text list "AlarmList": 1000 'F01000 - Внутрішня програмна помилка'; 1001 'F01001 - Виняток операції з плаваючою комою'; 1002 'F01002 - Внутрішня програмна помилка'; 1003 'F01003 - Затримка квитування під час доступу до пам’яті'; 1004 'N01004 (F, A) - Внутрішня програмна помилка'; 1005 'F01005 - Не вдалося завантажити прошивку компонента DRIVE-CLiQ'; 1006 'A01006 - Потрібне оновлення прошивки компонента DRIVE-CLiQ'; 1007 'A01007 - Потрібне повторне увімкнення живлення компонента DRIVE-CLiQ'; 1009 'A01009 (N) - CU: Перегрів модуля керування'; 1010 'F01010 - Невідомий тип приводу'; 1011 'F01011 (N) - Завантаження перервано'; 1012 'F01012 (N) - Помилка перетворення проєкту'; 1013 'A01013 - CU: Досягнуто або перевищено граничний ресурс вентилятора'; 1014 'F01014 - Топологія: змінено властивість компонента DRIVE-CLiQ'; 1015 'F01015 - Внутрішня програмна помилка'; 1016 'A01016 (F) - Змінено версію прошивки'; 1017 'A01017 - Змінено списки компонентів'; 1020 'A01020 - Не вдалося записати дані на RAM-диск'; 1023 'F01023 - Внутрішній програмний тайм-аут'; 1030 'F01030 - Відсутній сигнал справності головного керування'; 1031 'F01031 - Відсутній сигнал справності команди OFF у режимі REMOTE'; 1032 'A01032 (F) - ACX: Необхідно зберегти всі параметри'; 1033 'F01033 - Перемикання одиниць: некоректне опорне значення параметра'; 1034 'F01034 - Перемикання одиниць: не вдалося обчислити значення параметрів після зміни опорного значення'; 1035 'A01035 (F) - ACX: Пошкоджено файл резервної копії параметрів'; 1036 'F01036 (A) - ACX: Відсутній файл резервної копії параметрів'; 1038 'F01038 (A) - ACX: Не вдалося завантажити файл резервної копії параметрів'; 1039 'F01039 (A) - ACX: Не вдалося записати файл резервної копії параметрів'; 1040 'F01040 - Збережіть налаштування параметрів і виконайте повторне увімкнення живлення'; 1041 'F01041 - Потрібно зберегти параметри'; 1042 'F01042 - Помилка параметрів під час завантаження проєкту'; 1043 'F01043 - Критична помилка під час завантаження проєкту'; 1044 'F01044 - CU: Помилка описових даних'; 1045 'A01045 - CU: Некоректні конфігураційні дані'; 1049 'A01049 - CU: Не вдалося записати дані у файл'; 1050 'F01050 - Карта пам’яті несумісна з пристроєм'; 1054 'F01054 - CU: Перевищено системне обмеження'; 1055 'F01055 - CU: Внутрішня помилка (SYNO порту та прикладної програми не збігаються)'; 1056 'F01056 - CU: Внутрішня помилка (тактовий цикл групи параметрів уже призначено інакше)'; 1057 'F01057 - CU: Внутрішня помилка (інший тип DRIVE-CLiQ для підлеглого пристрою)'; 1058 'F01058 - CU: Внутрішня помилка (у топології відсутній підлеглий пристрій)'; 1059 'F01059 - CU: Внутрішня помилка (порт не існує)'; 1060 'F01060 - CU: Внутрішня помилка (група параметрів недоступна)'; 1061 'F01061 - CU: Внутрішня помилка (невідома прикладна програма)'; 1063 'F01063 - CU: Внутрішня помилка (PDM)'; 1064 'A01064 (F) - CU: Внутрішня помилка (CRC)'; 1068 'F01068 - CU: Переповнення пам’яті даних'; 1069 'A01069 - Несумісність резервної копії параметрів і пристрою'; 1070 'F01070 - Виконується завантаження проєкту/прошивки на карту пам’яті'; 1072 'F01072 - Карту пам’яті відновлено з резервної копії'; 1073 'A01073 (N) - Для резервної копії на карті пам’яті потрібне повторне увімкнення живлення'; 1082 'F01082 - Помилка параметрів під час увімкнення з резервної копії даних'; 1097 'A01097 (N) - Сервер NTP недоступний'; 1099 'A01099 (N) - Перевищено допуск синхронізації UTC'; 1100 'A01100 - CU: Карту пам’яті вилучено'; 1105 'F01105 (A) - CU: Недостатньо пам’яті'; 1106 'F01106 - CU: Недостатньо пам’яті'; 1107 'F01107 - CU: Не вдалося зберегти дані на карту пам’яті'; 1110 'F01110 - CU: До одного модуля керування підключено більше одного SINAMICS G'; 1111 'F01111 - CU: Змішана робота приводних модулів не допускається'; 1112 'F01112 - CU: Використання силового модуля не допускається'; 1120 'F01120 (A) - Не вдалося ініціалізувати термінал'; 1122 'F01122 (A) - Частота на вході вимірювального щупа занадто висока'; 1123 'F01123 - Силовий модуль не підтримує дискретні входи/виходи'; 1150 'F01150 - CU: Перевищено кількість екземплярів типу об’єкта приводу'; 1151 'F01151 - CU: Перевищено кількість об’єктів приводу заданої категорії'; 1152 'F01152 - CU: Некоректна комбінація типів об’єктів приводу'; 1200 'F01200 - CU: Внутрішня програмна помилка керування часовими квантами'; 1205 'F01205 - CU: Переповнення часового кванта'; 1221 'F01221 - CU: Базовий тактовий цикл занадто малий'; 1222 'F01222 - CU: Базовий тактовий цикл занадто малий (недостатньо часу на обробку зв’язку)'; 1223 'A01223 - CU: Некоректний час дискретизації'; 1224 'A01224 - CU: Некоректна частота імпульсів'; 1250 'F01250 - CU: Некоректні дані CU-EEPROM, доступні лише для читання'; 1251 'A01251 - CU: Некоректні дані читання/запису CU-EEPROM'; 1255 'F01255 - CU: Помилка даних EEPROM плати розширення, доступних лише для читання'; 1256 'A01256 - CU: Помилка даних читання/запису EEPROM плати розширення'; 1260 'F01260 - Програмне забезпечення не активоване'; 1275 'F01275 - Помилка опису обладнання'; 1276 'A01276 - Опис обладнання не повністю сумісний'; 1302 'A01302 - Помилка у трасуванні компонента'; 1303 'F01303 - Компонент виконує не підтримка потрібно функція'; 1304 'A01304 (F) - Версія прошивки компонента DRIVE-CLiQ застаріла'; 1305 'F01305 - Топологія: відсутній номер компонента'; 1306 'A01306 - Виконується оновлення прошивки компонента DRIVE-CLiQ'; 1314 'A01314 - Топологія: Компонент повинен не бути наявний'; 1317 'A01317 (N) - Деактивовано компонент повторно наявний'; 1318 'A01318 - BICO: наявні деактивовані міжз’єднання'; 1319 'A01319 - Встановлений компонент не ініціалізовано'; 1320 'A01320 - Топологія: номер об’єкта приводу відсутній у конфігурації'; 1321 'A01321 - Топологія: номер об’єкта приводу відсутній у конфігурації'; 1322 'A01322 - Топологія: номер об’єкта приводу двічі присутній у конфігурації'; 1323 'A01323 - Топологія: створено більше двох часткових списків'; 1324 'A01324 - Топологія: номер фіктивного об’єкта приводу створено некоректно'; 1325 'F01325 - Топологія: номер компонента відсутній у цільовій топології'; 1330 'A01330 - Топологія: швидке введення в експлуатацію неможливе'; 1331 'A01331 - Топологія: щонайменше один компонент не призначено об’єкту приводу'; 1340 'F01340 - Топологія: на одній лінії забагато компонентів'; 1341 'F01341 - Топологія: перевищено максимальну кількість компонентів DRIVE-CLiQ'; 1354 'F01354 - Топологія: фактична топологія містить неприпустимий компонент'; 1355 'F01355 - Топологія: Фактичний топологія змінено'; 1356 'F01356 - Топологія: виявлено несправний компонент DRIVE-CLiQ'; 1357 'F01357 - Топологія: на лінії DRIVE-CLiQ ідентифіковано два модулі керування'; 1358 'A01358 - Топологія: термінування лінії недоступне'; 1359 'F01359 - Топологія: продуктивність DRIVE-CLiQ недостатня'; 1360 'F01360 - Топологія: Фактичний топологія не допустимий'; 1361 'A01361 - Топологія: фактична топологія містить компоненти SINUMERIK і SIMOTION'; 1362 'A01362 - Топологія: порушено правило(а) топології'; 1375 'F01375 - Топологія: між двома компонентами дубльовано з’єднання'; 1380 'F01380 - Топологія: Фактичний топологія EEPROM несправний'; 1381 'A01381 - Топологія: силовий модуль встановлено некоректно'; 1382 'A01382 - Топологія: модуль датчика встановлено некоректно'; 1383 'A01383 - Топологія: термінальний модуль встановлено некоректно'; 1384 'A01384 - Топологія: модуль-концентратор DRIVE-CLiQ встановлено некоректно'; 1385 'A01385 - Топологія: модуль розширення контролера встановлено некоректно'; 1386 'A01386 - Топологія: компонент DRIVE-CLiQ встановлено некоректно'; 1389 'A01389 - Топологія: двигун із DRIVE-CLiQ встановлено некоректно'; 1416 'A01416 - Топологія: додатково встановлено компонент'; 1420 'A01420 - Топологія: Компонент інший'; 1425 'A01425 - Топологія: інший серійний номер'; 1428 'A01428 - Топологія: використано некоректне з’єднання'; 1451 'F01451 - Топологія: цільова топологія некоректна'; 1481 'A01481 (N) - Топологія: силовий модуль не підключено'; 1482 'A01482 - Топологія: модуль датчика не підключено'; 1483 'A01483 - Топологія: термінальний модуль не підключено'; 1484 'A01484 - Топологія: модуль-концентратор DRIVE-CLiQ не підключено'; 1485 'A01485 - Топологія: модуль розширення контролера не підключено'; 1486 'A01486 - Топологія: компонент DRIVE-CLiQ не підключено'; 1487 'A01487 - Топологія: компонент у слоті опцій не встановлено'; 1489 'A01489 - Топологія: двигун із DRIVE-CLiQ не підключено'; 1507 'A01507 (F, N) - BICO: наявні міжз’єднання з неактивними об’єктами'; 1508 'A01508 - BICO: перевищено кількість міжз’єднань з неактивними об’єктами'; 1510 'F01510 - BICO: джерело сигналу не має типу FLOAT'; 1511 'F01511 (A) - BICO: міжз’єднання з різними масштабуваннями'; 1512 'F01512 - BICO: масштабування недоступне'; 1513 'F01513 (N, A) - BICO: міжз’єднання між об’єктами приводу з різними масштабуваннями'; 1514 'A01514 (F) - BICO: помилка запису під час повторного з’єднання'; 1515 'F01515 (A) - BICO: запис до параметра не допускається, оскільки активне головне керування'; 1590 'A01590 (F) - Привід: перевищено інтервал технічного обслуговування двигуна'; 1600 'F01600 - SI P1 (CU): Ініційовано зупинку A'; 1611 'F01611 (A) - SI P1 (CU): Несправність у каналі контролю'; 1612 'F01612 - SI P1 (CU): Різні STO-входи силових модулів, підключених паралельно'; 1620 'N01620 (F, A) - SI P1 (CU): Безпечне вимкнення крутного моменту активний'; 1621 'N01621 (F, A) - SI P1 (CU): Активна безпечна зупинка 1'; 1625 'F01625 - SI P1 (CU): Помилка сигналу справності в даних безпеки'; 1630 'F01630 - SI P1 (CU): Гальмо керування помилка'; 1631 'A01631 (F, N) - SI P1 (CU): Конфігурація гальма утримання двигуна/SBC непрактична'; 1632 'F01632 - SI P1 (CU): Помилка сигналу керування/зворотного зв’язку запірного клапана'; 1640 'F01640 (N, A) - SI P1 (CU): Виявлено заміну компонента; потрібні квитування та збереження'; 1641 'F01641 (N, A) - SI P1 (CU): Виявлено заміну компонента; потрібне збереження'; 1649 'F01649 - SI P1 (CU): Внутрішня програмна помилка'; 1650 'F01650 - SI P1 (CU): Потрібне приймальне випробування'; 1651 'F01651 - SI P1 (CU): Не вдалося синхронізувати часові кванти безпеки'; 1652 'F01652 - SI P1 (CU): неприпустимий тактовий цикл контролю'; 1653 'F01653 - SI P1 (CU): PROFIBUS/PROFINET конфігурація помилка'; 1654 'A01654 (F, N) - SI P1 (CU): Відхилення конфігурації PROFIsafe'; 1655 'F01655 - SI P1 (CU): Узгодьте функції контролю'; 1656 'F01656 - SI CU: Помилка каналу 2 контролю параметрів'; 1657 'F01657 - SI P1 (CU): Некоректний номер телеграми PROFIsafe'; 1658 'F01658 - SI P1 (CU): Номери телеграм PROFIsafe відрізняються'; 1659 'F01659 - SI P1 (CU): Запит на запис параметра відхилено'; 1660 'F01660 - SI P1 (CU): Функції, пов’язані з безпекою, не підтримуються'; 1661 'F01661 - SI P1 (CU): Активна симуляція входів безпеки'; 1663 'F01663 - SI P1 (CU): Копіювання параметрів SI відхилено'; 1664 'F01664 - SI P1 (CU): Відсутнє автоматичне оновлення прошивки'; 1665 'F01665 - SI P1 (CU): Система несправна'; 1666 'A01666 (F) - SI Motion P1 (CU): Постійний сигнал «1» на F-DI для безпечного квитування'; 1669 'A01669 (F, N) - SI Motion: Несприятлива комбінація двигуна та силового модуля'; 1670 'F01670 - SI Motion: Некоректна параметризація модуля датчика'; 1671 'F01671 - SI Motion: Помилка параметризації енкодера'; 1672 'F01672 - SI P1 (CU): Програмне/апаратне забезпечення моторного модуля несумісне'; 1673 'F01673 - SI Motion: Програмне/апаратне забезпечення модуля датчика несумісне'; 1674 'F01674 - SI Motion P1 (CU): Функція безпеки не підтримується телеграмою PROFIsafe'; 1675 'F01675 - SI Motion P1: Налаштування у контролері PROFIBUS/PROFINET не допускаються'; 1679 'F01679 - SI CU: Змінено налаштування параметрів безпеки та топологію; потрібен теплий перезапуск/POWER ON'; 1680 'F01680 - SI Motion P1 (CU): Помилка контрольної суми функцій контролю безпеки'; 1681 'F01681 - SI Motion P1 (CU): Некоректне значення параметра'; 1682 'F01682 - SI Motion P1 (CU): Функція контролю не підтримується'; 1683 'F01683 - SI Motion P1 (CU): Відсутній дозвіл SOS/SLS'; 1684 'F01684 - SI Motion P1 (CU): Граничні значення безпечно обмеженого положення переплутано'; 1685 'F01685 - SI Motion P1 (CU): Граничне значення безпечно обмеженої швидкості занадто високе'; 1686 'F01686 - SI Motion: Некоректна параметризація кулачкового положення'; 1687 'F01687 - SI Motion: Некоректна параметризація модульного значення SCA (SN)'; 1688 'F01688 - SI Motion CU: Фактичний значення синхронізація не допустимий'; 1689 'C01689 - SI Motion: Вісь повторно сконфігуровано'; 1690 'F01690 - SI Motion: Помилка збереження даних у NVRAM'; 1691 'A01691 (F) - SI Motion: Значення Ti та To непридатні для циклу DP'; 1692 'F01692 - SI Motion P1 (CU): Значення параметра не допускається для режиму без енкодера'; 1693 'A01693 (F) - SI P1 (CU): Змінено налаштування параметрів безпеки; потрібен теплий перезапуск/повторне увімкнення живлення'; 1694 'F01694 (A) - SI Motion CU: Версія прошивки моторного/гідравлічного модуля старіша за версію модуля керування'; 1695 'A01695 (F) - SI Motion: Модуль датчика замінено'; 1696 'A01696 (F) - SI Motion: Під час завантаження вибрано тестову зупинку для функцій контролю руху'; 1697 'A01697 (F) - SI Motion: Потрібна тестова зупинка для функцій контролю руху'; 1698 'A01698 (F) - SI P1 (CU): Активний режим введення в експлуатацію'; 1699 'A01699 (F) - SI P1 (CU): Потрібна тестова зупинка для STO'; 1700 'C01700 - SI Motion P1 (CU): Ініційовано зупинку A'; 1701 'C01701 - SI Motion P1 (CU): Ініційовано зупинку B'; 1706 'C01706 - SI Motion P1 (CU): Перевищено обмеження SAM/SBR'; 1707 'C01707 - SI Motion P1 (CU): Перевищено допуск для безпечної робочої зупинки'; 1708 'C01708 - SI Motion P1 (CU): Ініційовано зупинку C'; 1709 'C01709 - SI Motion P1 (CU): Ініційовано зупинку D'; 1710 'C01710 - SI Motion P1 (CU): Ініційовано зупинку E'; 1711 'C01711 - SI Motion P1 (CU): Несправність у каналі контролю'; 1712 'C01712 - SI Motion P1 (CU): Несправність обробки F-IO'; 1714 'C01714 - SI Motion P1 (CU): Безпечно обмежена швидкість перевищено'; 1715 'C01715 - SI Motion P1 (CU): Безпечно обмежене положення перевищено'; 1716 'C01716 - SI Motion P1 (CU): Перевищено допуск для безпечного напрямку руху'; 1717 'C01717 - SI Motion P1 (CU): Перевищено обмеження SLA'; 1730 'C01730 - SI Motion P1 (CU): Некоректний опорний блок для динамічної безпечно обмеженої швидкості'; 1745 'C01745 - SI Motion P1 (CU): Перевірка гальмівного моменту для тесту гальма'; 1750 'C01750 - SI Motion P1 (CU): Апаратна несправність енкодера, важливого для безпеки'; 1751 'C01751 - SI Motion P1 (CU): Несправність перевірки ефективності енкодера, важливого для безпеки'; 1752 'C01752 - SI Motion P1 (CU): Некоректне референтне положення'; 1770 'C01770 - SI Motion P1 (CU): Помилка розбіжності відмовобезпечних входів/виходів'; 1772 'A01772 - SI Motion P1 (CU): Виконується тестова зупинка для відмовобезпечних дискретних виходів'; 1773 'F01773 - SI Motion P1 (CU): Помилка тестової зупинки відмовобезпечного дискретного виходу'; 1774 'A01774 - SI Motion P1 (CU): Потрібна тестова зупинка для відмовобезпечних дискретних виходів'; 1780 'A01780 - За вибору SBT гальмо замкнене'; 1781 'A01781 - Перевищено час розгальмовування гальма SBT'; 1782 'A01782 - SBT гальмо тест некоректний керування'; 1783 'A01783 - Перевищено час загальмовування гальма SBT'; 1784 'A01784 - Тест гальма SBT скасовано через несправність'; 1785 'A01785 - Помилка конфігурації тесту гальма SBT'; 1786 'F01786 - Змінено джерело сигналу SCC'; 1787 'F01787 - Інший тип двигуна SBT'; 1788 'A01788 - SI: Автоматична тестова зупинка очікує скасування вибору STO через функції контролю руху'; 1789 'A01789 - SI: Автоматична тестова зупинка та тест гальма не допускаються, коли вибрано тестову зупинку'; 1794 'A01794 (N) - SI Motion: Перевірка модульного значення для безпечного положення через PROFIsafe'; 1795 'A01795 - SI Motion P1 (CU): Перевищено час очікування після виходу зі скасування безпечних імпульсів'; 1796 'A01796 (F, N) - SI P1 (CU): Очікування зв’язку'; 1797 'C01797 - SI Motion P1 (CU): Вісь не пройшла безпечне реферування'; 1798 'C01798 - SI Motion P1 (CU): Тест зупинка для рух контроль функції виконується'; 1799 'C01799 - SI Motion P1 (CU): Приймальне тест режим активний'; 1800 'F01800 (A) - DRIVE-CLiQ: помилка обладнання/конфігурації'; 1839 'A01839 - Діагностика DRIVE-CLiQ: несправність кабелю до компонента'; 1840 'A01840 - SMI: Компонент виявлено без Дані двигуна'; 1900 'A01900 (F) - PB/PN: Конфігурація Помилка телеграми'; 1902 'A01902 - PB/PN: параметризація синхронної роботи за тактовим циклом не допускається'; 1903 'A01903 (F) - COMM INT: Приймання конфігурація дані некоректний'; 1910 'F01910 (N, A) - Польова шина: тайм-аут заданого значення'; 1911 'F01911 (N, A) - PB/PN: відмова тактового циклу синхронної роботи'; 1912 'F01912 (N, A) - PB/PN: відмова сигналу справності синхронної роботи за тактовим циклом'; 1913 'F01913 (N, A) - COMM INT: закінчився контрольний час сигналу справності'; 1914 'F01914 (N, A) - COMM INT: Контроль час конфігурація закінчився'; 1915 'F01915 (N, A) - PB/PN: відмова сигналу справності синхронної роботи за тактовим циклом, об’єкт приводу 1'; 1920 'A01920 (F) - PROFIBUS: перервано циклічне з’єднання'; 1921 'A01921 (F) - PROFIBUS: приймання заданих значень після To'; 1925 'A01925 (F) - Modbus TCP: з’єднання перервано'; 1930 'A01930 - PB/PN: час дискретизації регулятора струму не дорівнює синхронному тактовому циклу'; 1931 'A01931 - PB/PN: час дискретизації регулятора швидкості не дорівнює синхронному тактовому циклу'; 1932 'A01932 - PB/PN: відсутня синхронізація тактового циклу для DSC'; 1940 'A01940 - PB/PN: синхронізм тактового циклу не досягнуто'; 1941 'A01941 - PB/PN: відсутній сигнал тактового циклу під час встановлення зв’язку по шині'; 1943 'A01943 - PB/PN: помилка сигналу тактового циклу під час встановлення зв’язку по шині'; 1944 'A01944 - PB/PN: синхронізм сигналу справності не досягнуто'; 1945 'A01945 - PROFIBUS: З’єднання до Видавець не вдалося виконати'; 1946 'F01946 (A) - PROFIBUS: з’єднання з видавцем перервано'; 1950 'F01950 (N, A) - PB/PN: не вдалося синхронізувати синхронну роботу за тактовим циклом'; 1951 'F01951 - CU SYNC: відсутній тактовий цикл прикладної синхронізації'; 1952 'F01952 - CU DRIVE-CLiQ: синхронізація компонента не підтримується'; 1953 'A01953 - CU SYNC: синхронізацію не завершено'; 1954 'F01954 - CU DRIVE-CLiQ: не вдалося виконати синхронізацію'; 1955 'A01955 - CU DRIVE-CLiQ: синхронізацію об’єкта приводу не завершено'; 1970 'A01970 - CBExx: циклічне з’єднання перервано'; 1971 'A01971 - CBExx: перевищено максимальну кількість контролерів'; 1977 'A01977 (N) - CBE41: перегрів аварійне повідомлення'; 1978 'F01978 (N, A) - CBE41: перегрів несправність'; 1979 'A01979 - CBExx: внутрішня помилка циклічної передачі даних'; 1980 'A01980 - PN: циклічний з’єднання перервано'; 1981 'A01981 - PN: Максимальний номер з контролери перевищено'; 1982 'A01982 - PN: секунда регулятор відсутній'; 1983 'A01983 - PN: виконується перемикання системної резервованості'; 1989 'A01989 - PN: внутрішній Помилка циклічної передачі даних'; 1990 'A01990 (F) - USS: PZD конфігурація помилка'; 2000 'A02000 - Функціональний генератор: пуск неможливий'; 2005 'A02005 - Функціональний генератор: привід не існує'; 2006 'A02006 - Функціональний генератор: для з’єднання не задано привід'; 2007 'A02007 - Функціональний генератор: привід не належить до типу SERVO/VECTOR/DC_CTRL'; 2008 'A02008 - Функціональний генератор: привід задано кілька разів'; 2009 'A02009 - Функціональний генератор: неприпустимий режим'; 2010 'A02010 - Функціональний генератор: задане значення швидкості приводу не дорівнює нулю'; 2011 'A02011 - Функціональний генератор: фактична швидкість приводу не дорівнює нулю'; 2015 'A02015 - Функціональний генератор: відсутні сигнали дозволу приводу'; 2016 'A02016 - Функціональний генератор: виконується намагнічування'; 2020 'A02020 - Функціональний генератор: параметр неможливо змінити'; 2025 'A02025 - Функціональний генератор: період занадто короткий'; 2026 'A02026 - Функціональний генератор: тривалість імпульсу занадто велика'; 2030 'A02030 - Функціональний генератор: фізична адреса дорівнює нулю'; 2040 'A02040 - Функціональний генератор: неприпустиме значення зміщення'; 2041 'A02041 - Функціональний генератор: неприпустиме значення смуги пропускання'; 2047 'A02047 - Функціональний генератор: некоректний тактовий цикл часового кванта'; 2050 'A02050 - Трасування: пуск неможливий'; 2051 'A02051 - Трасування: реєстрація неможлива через захист ноу-хау'; 2055 'A02055 - Трасування: час реєстрації занадто короткий'; 2056 'A02056 - Трасування: цикл реєстрації занадто короткий'; 2057 'A02057 - Трасування: некоректний тактовий цикл часового кванта'; 2058 'A02058 - Трасування: некоректний тактовий цикл часового кванта для безперервного трасування'; 2059 'A02059 - Трасування: некоректний тактовий цикл часового кванта для 2×8 каналів реєстрації'; 2060 'A02060 - Трасування: відсутній сигнал для трасування'; 2061 'A02061 - Трасування: Некоректний сигнал'; 2062 'A02062 - Трасування: Некоректний запуск сигнал'; 2063 'A02063 - Трасування: некоректний тип даних'; 2070 'A02070 - Трасування: Параметр не може бути змінено'; 2075 'A02075 - Трасування: час передтригера занадто великий'; 2080 'F02080 - Трасування: параметризацію видалено через перемикання одиниць'; 2085 'A02085 - Повідомлення функція: Параметризація помилка'; 2095 'A02095 - MTRACE 0: кілька трасування не може бути активовано'; 2096 'A02096 - MTRACE 0: не може бути збережено'; 2097 'A02097 - MTRACE 1: кілька трасування не може бути активовано'; 2098 'A02098 - MTRACE 1: не може бути збережено'; 2099 'A02099 - Трасування: Недостатній Керування Модуль пам’ять'; 2100 'A02100 - Привід: час обчислення регулятора струму занадто короткий'; 2150 'A02150 - TEC: Технологія Розширення не може бути завантажено'; 2151 'F02151 (A) - TEC: Внутрішня програмна помилка'; 2152 'F02152 (A) - TEC: недостатній пам’ять'; 2153 'F02153 - TEC: технологія функція виконує не існує'; 3000 'F03000 - Несправність NVRAM під час виконання дії'; 3001 'F03001 - NVRAM контрольна сума некоректний'; 3500 'F03500 (A) - TM: Ініціалізація'; 3501 'A03501 - TM: зміна часу дискретизації'; 3505 'F03505 (N, A) - CU: Аналоговий вхід провід обрив'; 3506 'A03506 (F, N) - Відсутнє живлення 24 В'; 3507 'A03507 (F, N) - Дискретний вихід не встановлено'; 3510 'A03510 (F, N) - CU: Калібрування дані не правдоподібний'; 3550 'A03550 - TM: Швидкість задане фільтр власний частота > Найквіста частота'; 3590 'F03590 (N, A) - TM: Модуль не готовий'; 5000 'A05000 (N) - Силовий модуль: перегрів радіатора інвертора AC'; 5001 'A05001 (N) - Силовий модуль: перегрів кристала запірного шару'; 5002 'A05002 (N) - Силовий модуль: перегрів повітря на вході'; 5003 'A05003 (N) - Силовий модуль: внутрішній перегрів'; 5004 'A05004 (N) - Силовий модуль: перегрів випрямляча'; 5005 'A05005 - Охолоджувальний агрегат: Охолодження середовище витрата витрата занадто низький'; 5006 'A05006 (N) - Силовий модуль: перегрів за тепловою моделлю'; 5007 'N05007 (A) - Силовий модуль: перегрів за тепловою моделлю (шасі PU)'; 5050 'F05050 - Паралельне коло: дозвіл імпульсів за наявності заборони імпульсів'; 5051 'F05051 - Паралельне коло: Відсутній дозвіл імпульсів силового модуля'; 5052 'A05052 (F) - Паралельне коло: неприпустима асиметрія струму'; 5053 'A05053 (F) - Паралельне коло: неприпустима асиметрія напруги кола постійного струму'; 5054 'A05054 (N) - Паралельне коло: Силовий модуль деактивовано'; 5055 'F05055 - Паралельне з’єднання: силові модулі з неприпустимими кодовими номерами'; 5056 'F05056 - Паралельне коло: версії EEPROM силових модулів відрізняються'; 5057 'F05057 - Паралельне коло: версії прошивки силових модулів відрізняються'; 5058 'F05058 - Паралельне коло: версії EEPROM VSM відрізняються'; 5059 'F05059 - Паралельне коло: версії прошивки VSM відрізняються'; 5060 'F05060 - Паралельне коло: Версія прошивки силового модуля не збігається'; 5061 'F05061 - Кількість VSM на вводі'; 5064 'F05064 - Паралельне з’єднання: Імпульс синхронізація помилка'; 5065 'A05065 (F, N) - Напруга виміряний значення не правдоподібний'; 5066 'A05066 (F, N) - Паралельне з’єднання: неприпустима асиметрія напруги VSM'; 5118 'F05118 (A) - Перевищено час контролю одночасності контактора попереднього заряду'; 5119 'F05119 (A) - Перевищено час контролю одночасності байпасного контактора'; 6000 'F06000 - Ввід: Попередній заряд контроль час закінчився'; 6010 'F06010 - Ввід: у роботі відсутній силовий модуль EP 24 В'; 6050 'F06050 - Ввід: режим Smart не підтримується'; 6052 'F06052 - Ввід: Фільтр температура обробка не підтримується'; 6080 'F06080 (A) - Ввід: параметр помилка'; 6100 'F06100 - Ввід: Вимкнення через до мережа Занижена напруга живлення умова'; 6105 'A06105 (F) - Ввід: Мережа Занижена напруга живлення'; 6200 'F06200 - Ввід: відсутня одна або кілька фаз мережі'; 6205 'A06205 (F) - Ввід: провал напруги щонайменше в одній фазі мережі'; 6206 'A06206 (F) - Ввід: аварійне повідомлення про асиметрію струмів мережі'; 6207 'F06207 (N, A) - Ввід: асиметрія струмів мережі'; 6208 'A06208 (F, N) - Лінія вводу: асиметрія напруги живлення'; 6210 'F06210 - Ввід: Сумування струм занадто високий'; 6211 'F06211 - Ввід: сумарний струм неприпустимо високий'; 6215 'A06215 (F) - Ввід: Сумування струм занадто високий'; 6250 'A06250 (F, N) - Ввід: несправний(і) конденсатор(и) щонайменше в одній фазі мережевого фільтра'; 6255 'F06255 (A) - Ввід: температура поріг значення не допустимий'; 6260 'A06260 - Ввід: Температура у мережа фільтр занадто високий'; 6261 'F06261 - Ввід: температура мережевого фільтра постійно занадто висока'; 6262 'F06262 - Ввід: Температура вимикач у мережа фільтр відкритий коли перемикання на'; 6300 'F06300 - Ввід: напруга мережі занадто висока на POWER ON'; 6301 'A06301 (F) - Ввід: перенапруга мережі'; 6310 'F06310 (A) - Ввід: напругу живлення (p0210) параметризовано некоректно'; 6311 'F06311 - Ввід: некоректна напруга живлення (p0210)'; 6320 'F06320 - Головний/підлеглий: некоректне керування 4-канальним мультиплексором'; 6321 'F06321 - Головний/підлеглий: некоректне керування 6-канальним мультиплексором'; 6350 'A06350 (F) - Ввід: Виміряний Частота мережі занадто висока'; 6351 'A06351 (F) - Ввід: Виміряний Частота мережі занадто низька'; 6400 'A06400 - Ввід: вибрано/активовано ідентифікацію даних мережі'; 6401 'A06401 - Ввід: вибрано/активовано ідентифікацію даних трансформатора/тестовий режим'; 6500 'F06500 - Ввід: синхронізація з мережею неможлива'; 6502 'A06502 (F, N) - Ввід: не вдалося синхронізуватися з мережею під час намагнічування трансформатора'; 6503 'F06503 - Ввід: чорний пуск мережі не вдався'; 6504 'F06504 - Ввід: не вдалося синхронізувати синхронну автономну мережу'; 6505 'F06505 - Ввід: для намагнічування трансформатора перевищено обмеження струму'; 6601 'A06601 (F) - Ввід: Струм зміщення вимірювання перервано'; 6602 'A06602 (F) - Ввід: вимірювання зміщення струму неможливе'; 6700 'F06700 (A) - Ввід: Вимикач мережа контактор для навантаження умова'; 6800 'A06800 (F) - Ввід: досягнуто максимальної усталеної напруги кола постійного струму'; 6810 'A06810 (F) - Ввід: напруга кола постійного струму опустилася нижче порога аварійного повідомлення'; 6849 'A06849 (F, N) - Ввід: Коротке замикання робота активний'; 6850 'F06850 - Ввід: коротке замикання триває надто довго'; 6851 'F06851 - Ввід: спрацював контроль розподіленої лінії вводу'; 6855 'F06855 - Ввід: Мережа фільтр контролювати спрацював'; 6860 'A06860 - Ввід: активація функціонального модуля неможлива'; 6900 'A06900 (F) - Гальмівний Модуль: Несправність (1 -> 0)'; 6901 'A06901 - Модуль гальмування: попереднє вимкнення за I²t'; 6904 'A06904 (N) - Внутрішня функція модуля гальмування заблокована'; 6905 'A06905 - Гальмівний Модуль внутрішній I²t вимкнення аварійне повідомлення'; 6906 'F06906 (A) - Гальмівний Модуль внутрішній несправність'; 6907 'F06907 - Гальмівний Модуль Внутрішній перегрів'; 6908 'F06908 - Гальмівний Модуль Внутрішній перегрів вимкнення'; 6909 'F06909 - Внутрішня несправність Vce модуля гальмування'; 6921 'A06921 (N) - Гальмівний резистор фаза асиметрія'; 6922 'F06922 - Гальмівний резистор Відсутня фаза'; 7011 'F07011 - Привід: перегрів двигуна'; 7012 'A07012 (N) - Привід: Двигун температура модель 1/3 перегрів'; 7013 'F07013 - Привід: Двигун температура модель конфігурація несправність'; 7014 'A07014 (N) - Привід: Двигун температура модель конфігурація аварійне повідомлення'; 7015 'A07015 - Привід: Датчик температури двигуна аварійне повідомлення'; 7016 'F07016 - Привід: Несправність датчика температури двигуна'; 7017 'A07017 - Перевищено додатковий поріг аварійного повідомлення за температурою'; 7018 'F07018 - Перевищено додатковий поріг несправності за температурою'; 7048 'F07048 - Привід: Некоректний характеристика вимірювання'; 7080 'F07080 - Привід: Некоректний керування параметр'; 7082 'F07082 - Макрос: виконання неможливе'; 7083 'F07083 - Макрос: ACX файл не виявлено'; 7084 'F07084 - Макрос: умову WaitUntil не виконано'; 7085 'F07085 - Привід: змінено параметри розімкненого/замкненого керування'; 7086 'F07086 - Перемикання одиниць: порушення обмеження параметра через зміну опорного значення'; 7087 'F07087 - Привід: бездатчиковий режим неможливий для вибраної частоти імпульсів'; 7088 'F07088 - Перемикання одиниць: порушення обмеження параметра через перемикання одиниць'; 7089 'A07089 - Перемикання одиниць: активацію функціонального модуля заблоковано через перемикання одиниць'; 7090 'F07090 - Привід: верхня межа крутного моменту менша за нижню'; 7091 'A07091 - Привід: некоректно визначено динамічну характеристику регулятора струму'; 7092 'A07092 - Привід: оцінювач моменту інерції ще не готовий'; 7093 'F07093 (A) - Привід: Тест сигнал помилка'; 7094 'A07094 - Загальне порушення обмеження параметра'; 7095 'A07095 (N) - Привід: активовано One Button Tuning'; 7097 'F07097 (A) - Привід: обмеження відстані помилки тестового сигналу'; 7098 'F07098 (A) - Привід: помилка конфігурації One Button Tuning'; 7100 'F07100 - Привід: неможливо скинути часи дискретизації'; 7110 'F07110 - Привід: часи дискретизації та базовий тактовий цикл не збігаються'; 7140 'A07140 - Привід: час дискретизації регулятора струму для шпинделя не збігається'; 7200 'A07200 - Привід: наявна команда ON головного керування'; 7220 'F07220 (N, A) - Привід: Відсутнє головне керування від PLC'; 7300 'F07300 (A) - Привід: Мережа контактор зворотний зв’язок сигнал відсутній'; 7311 'F07311 - Байпас двигун вимикач'; 7312 'F07312 - Байпасний вимикач зі сторони мережі:'; 7320 'F07320 - Привід: Автоматичний перезапуск перервано'; 7321 'A07321 - Привід: Автоматичний перезапуск активний'; 7329 'A07329 (N) - Привід: не працює оцінювач kT, характеристика kT(iq) або компенсація напруги'; 7330 'F07330 - Підхоплення обертового двигуна: виміряний пошуковий струм занадто малий'; 7331 'F07331 - На льоту перезапуск: Функція не підтримується'; 7332 'N07332 - Підхоплення обертового двигуна: максимальну швидкість зменшено'; 7333 'F07333 - Функція замкненого керування не підтримується'; 7334 'F07334 (N, A) - Функція неможлива'; 7350 'A07350 (F) - Привід: вимірювальний щуп параметризовано на дискретний вихід'; 7351 'A07351 (F) - Привід: вимірювальний щуп параметризовано на дискретний вихід'; 7354 'A07354 - Привід: компенсація зубчастого моменту неможлива'; 7355 'F07355 (N, A) - Привід: помилка під час навчання компенсації зубчастого моменту'; 7356 'A07356 (N) - Привід: Зубчастість крутний момент компенсація двигун або енкодер послідовний номер інший'; 7400 'A07400 (N) - Привід: активний регулятор максимальної напруги кола постійного струму'; 7401 'A07401 (N) - Привід: регулятор максимальної напруги кола постійного струму деактивовано'; 7402 'A07402 (N) - Привід: активний регулятор мінімальної напруги кола постійного струму'; 7403 'F07403 (N, A) - Привід: досягнуто нижнього порога напруги кола постійного струму'; 7404 'F07404 - Привід: досягнуто верхнього порога напруги кола постійного струму'; 7405 'F07405 (N, A) - Привід: швидкість кінетичного буферування опустилася нижче мінімальної'; 7406 'F07406 (N, A) - Привід: перевищено максимальний час кінетичного буферування'; 7407 'F07407 - Привід: зниження Vdc не допускається'; 7409 'A07409 (N) - Привід: керування U/f, активний регулятор обмеження струму'; 7410 'F07410 - Привід: Струм регулятор вихід обмежений'; 7411 'F07411 - Привід: Потік регулятор вихід обмежений'; 7412 'F07412 - Привід: некоректний кут комутації (модель двигуна)'; 7413 'F07413 - Привід: некоректний кут комутації (ідентифікація положення полюса)'; 7414 'F07414 (N, A) - Привід: Змінено серійний номер енкодера'; 7415 'N07415 (F) - Привід: Кутовий комутація зміщення передавання виконується'; 7416 'A07416 - Привід: Потік регулятор конфігурація'; 7417 'F07417 - Привід: метод імпульсного керування неправдоподібний (модель двигуна)'; 7419 'F07419 - Привід: помилка адаптації фільтра заданого значення струму'; 7420 'F07420 - Привід: Струм задане фільтр власний частота > Найквіста частота'; 7421 'F07421 - Привід: Швидкість фільтр власний частота > Найквіста частота'; 7422 'F07422 - Привід: Опорний модель власний частота > Найквіста частота'; 7423 'F07423 - Привід: APC фільтр власний частота > Найквіста частота'; 7424 'A07424 - Привід: умова роботи для APC некоректна'; 7425 'F07425 - Привід: APC контроль час для швидкість обмеження закінчився'; 7426 'F07426 (A) - Технологія регулятор фактичний значення обмежений'; 7428 'A07428 (N) - Помилка параметризації технологічного регулятора'; 7429 'F07429 - Привід: DSC без енкодера неможлива'; 7430 'F07430 - Привід: перемикання на розімкнене керування крутним моментом неможливе'; 7431 'F07431 - Привід: перемикання на бездатчиковий режим неможливе'; 7432 'F07432 - Привід: двигун без захисту від перенапруги'; 7433 'F07433 - Привід: замкнене керування з енкодером неможливе, оскільки енкодер не розпарковано'; 7434 'F07434 - Привід: неможливо змінити напрямок обертання за ввімкнених імпульсів'; 7435 'F07435 (N) - Привід: налаштування генератора рампової функції для бездатчикового векторного керування'; 7439 'F07439 - Привід: Функція не підтримується'; 7440 'A07440 - EPOS: час ривка обмежено'; 7441 'A07441 - LR: збережіть зміщення положення налаштування абсолютного енкодера'; 7442 'F07442 (A) - LR: багатообертовий режим не відповідає модульному діапазону'; 7443 'F07443 (A) - LR: Координата референтної точки поза допустимим діапазоном'; 7446 'F07446 (A) - Навантаження шестерня: Неможливо скинути супроводження положення'; 7447 'F07447 - Навантаження шестерня: Положення супроводження, максимальний фактичний значення перевищено'; 7448 'F07448 (A) - Редуктор навантаження: лінійна вісь під час супроводження положення перевищила максимальний діапазон'; 7449 'F07449 (A) - Навантаження шестерня: Положення супроводження фактичний положення поза допуск вікно'; 7450 'F07450 (A) - LR: спрацював контроль зупинки'; 7451 'F07451 (A) - LR: Положення контроль має спрацював'; 7452 'F07452 (A) - LR: похибка слідкування занадто велика'; 7453 'F07453 - LR: Помилка попередньої обробки фактичного значення положення'; 7454 'A07454 - LR: Для попередньої обробки фактичного значення положення відсутній коректний енкодер'; 7455 'A07455 - EPOS: обмежено максимальну швидкість'; 7456 'A07456 - EPOS: обмежено задану швидкість'; 7457 'A07457 - EPOS: Комбінація з вхід сигнали не допускається'; 7458 'F07458 - EPOS: Опорний кулачковий не виявлено'; 7459 'F07459 - EPOS: Відсутній нульовий мітка'; 7460 'F07460 - EPOS: Кінець з опорний кулачковий не виявлено'; 7461 'A07461 - EPOS: референтну точку не задано'; 7462 'A07462 - EPOS: вибраний номер блоку переміщення не існує'; 7463 'A07463 (F) - EPOS: у блоці переміщення не запитано зовнішню зміну блоку'; 7464 'F07464 - EPOS: блок переміщення некоректний'; 7465 'A07465 - EPOS: блок переміщення не має наступного блоку'; 7466 'A07466 - EPOS: номер блоку переміщення призначено кілька разів'; 7467 'A07467 - EPOS: блок переміщення має неприпустимі параметри завдання'; 7468 'A07468 - EPOS: ціль переходу блоку переміщення не існує'; 7469 'A07469 - EPOS: цільове положення блоку переміщення нижче від’ємного програмного кінцевого вимикача'; 7470 'A07470 - EPOS: цільове положення блоку переміщення вище додатного програмного кінцевого вимикача'; 7471 'A07471 - EPOS: цільове положення блоку переміщення поза модульним діапазоном'; 7472 'A07472 - EPOS: ABS_POS/ABS_NEG для блоку переміщення неможливе'; 7473 'A07473 (F) - EPOS: досягнуто початку діапазону переміщення'; 7474 'A07474 (F) - EPOS: досягнуто кінця діапазону переміщення'; 7475 'F07475 (A) - EPOS: цільове положення нижче початку діапазону переміщення'; 7476 'F07476 (A) - EPOS: цільове положення вище кінця діапазону переміщення'; 7477 'A07477 (F) - EPOS: Цільовий положення < програмне забезпечення обмеження вимикач мінус'; 7478 'A07478 (F) - EPOS: Цільовий положення > програмне забезпечення обмеження вимикач плюс'; 7479 'A07479 - EPOS: Програмне забезпечення обмеження вимикач мінус досягнуто'; 7480 'A07480 - EPOS: Програмне забезпечення обмеження вимикач плюс досягнуто'; 7481 'F07481 (A) - EPOS: Вісь положення < програмне забезпечення обмеження вимикач мінус'; 7482 'F07482 (A) - EPOS: Вісь положення > програмне забезпечення обмеження вимикач плюс'; 7483 'A07483 - EPOS: під час руху до жорсткого упора не досягнуто затискного моменту'; 7484 'F07484 - EPOS: Фіксований зупинка поза контроль вікно'; 7485 'F07485 (A) - EPOS: Фіксований зупинка не досягнуто'; 7486 'A07486 - EPOS: відсутня проміжна зупинка'; 7487 'A07487 - EPOS: відсутнє відхилення завдання переміщення'; 7488 'F07488 - EPOS: відносне позиціонування неможливе'; 7489 'A07489 - EPOS: корекція референтної точки поза вікном'; 7490 'F07490 (N) - EPOS: під час переміщення знято сигнал дозволу'; 7491 'F07491 (A) - EPOS: STOP кулачковий мінус досягнуто'; 7492 'F07492 (A) - EPOS: STOP кулачковий плюс досягнуто'; 7493 'F07493 - LR: переповнення діапазону значень фактичного положення'; 7494 'F07494 - LR: Виконується перемикання набору даних приводу'; 7495 'A07495 (F, N) - LR: Функцію реферування перервано'; 7496 'A07496 - EPOS: дозвіл неможливий'; 7497 'A07497 (N) - LR: Активовано значення налаштування положення'; 7498 'A07498 (F) - LR: Обробка вимірювального щупа неможлива'; 7499 'F07499 (A) - EPOS: кулачок реверсу досягнуто за неправильного напрямку переміщення'; 7500 'F07500 - Привід: набір даних силового модуля PDS не налаштовано'; 7501 'F07501 - Привід: набір даних двигуна MDS не налаштовано'; 7502 'F07502 - Привід: набір даних енкодера EDS не налаштовано'; 7503 'F07503 - EPOS: кулачок STOP досягнуто за неправильного напрямку переміщення'; 7504 'A07504 - Привід: набір даних двигуна не призначено набору даних приводу'; 7505 'A07505 - EPOS: завдання руху до жорсткого упора неможливе у режимі U/f/SLVC'; 7506 'A07506 - EPOS: перевірте BICO-міжз’єднання між EPOS і регулятором положення'; 7507 'A07507 - EPOS: неможливо встановити референтну точку'; 7509 'F07509 - Привід: відсутнє призначення компонента'; 7510 'F07510 - Привід: однаковий енкодер у наборі даних приводу'; 7511 'F07511 - Привід: енкодер використано кілька разів'; 7512 'F07512 - Привід: неможливо параметризувати перемикання набору даних енкодера'; 7514 'A07514 (N) - Привід: структура даних не відповідає інтерфейсному модулю'; 7515 'F07515 - Привід: силовий модуль і двигун підключено некоректно'; 7516 'F07516 - Привід: виконайте повторне введення в експлуатацію набору даних'; 7517 'F07517 - Привід: перемикання набору даних енкодера параметризовано некоректно'; 7518 'F07518 - Привід: перемикання набору даних двигуна параметризовано некоректно'; 7519 'A07519 - Привід: перемикання двигуна параметризовано некоректно'; 7520 'A07520 - Привід: неможливо перемкнути двигун'; 7530 'A07530 - Привід: набір даних приводу DDS відсутній'; 7531 'A07531 - Привід: набір даних команд CDS відсутній'; 7532 'A07532 (N) - Привід: бездатчикове керування не введено в експлуатацію'; 7541 'A07541 - Привід: перемикання набору даних неможливе'; 7550 'A07550 (F, N) - Привід: неможливо скинути параметри енкодера'; 7551 'F07551 - Привід енкодер: Відсутній комутація кут інформація'; 7552 'F07552 (A) - Привід енкодер: Енкодер конфігурація не підтримується'; 7553 'F07553 (A) - Привід енкодер: Модуль датчика конфігурація не підтримується'; 7555 'F07555 (A) - Привід енкодер: Конфігурація положення супроводження'; 7556 'F07556 - Вимірювальна шестерня: перевищено максимальне фактичне значення під час супроводження положення'; 7557 'A07557 (F) - Енкодер 1: Координата референтної точки поза допустимим діапазоном'; 7558 'A07558 (F) - Енкодер 2: Координата референтної точки поза допустимим діапазоном'; 7559 'A07559 (F) - Енкодер 3: Координата референтної точки поза допустимим діапазоном'; 7560 'F07560 - Привід енкодер: Номер з імпульси є не до потужність з два'; 7561 'F07561 - Привід енкодер: Номер з багатообертовий імпульси є не до потужність з два'; 7562 'F07562 (A) - Привід, енкодер: супроводження положення інкрементального енкодера неможливе'; 7563 'F07563 (A) - Привід енкодер: XIST1_ERW конфігурація некоректний'; 7565 'A07565 (F, N) - Привід: помилка енкодера в інтерфейсі енкодера PROFIdrive 1'; 7566 'A07566 (F, N) - Привід: помилка енкодера в інтерфейсі енкодера PROFIdrive 2'; 7567 'A07567 (F, N) - Привід: помилка енкодера в інтерфейсі енкодера PROFIdrive 3'; 7569 'A07569 (F) - Активна ідентифікація енкодера'; 7570 'N07570 (F) - Енкодер ідентифікація дані передавання виконується'; 7575 'F07575 - Привід: Двигун енкодер не готовий'; 7576 'A07576 - Привід: Без енкодера робота через до несправність активний'; 7577 'A07577 (F) - Енкодер 1: Обробка вимірювального щупа неможлива'; 7578 'A07578 (F) - Енкодер 2: Обробка вимірювального щупа неможлива'; 7579 'A07579 (F) - Енкодер 3: Обробка вимірювального щупа неможлива'; 7580 'A07580 (F, N) - Привід: відсутній модуль датчика з відповідним номером компонента'; 7581 'A07581 (F) - Енкодер 1: Помилка попередньої обробки фактичного значення положення'; 7582 'A07582 (F) - Енкодер 2: Помилка попередньої обробки фактичного значення положення'; 7583 'A07583 (F) - Енкодер 3: Помилка попередньої обробки фактичного значення положення'; 7584 'A07584 - Енкодер 1: Активовано значення налаштування положення'; 7585 'A07585 - Енкодер 2: Активовано значення налаштування положення'; 7586 'A07586 - Енкодер 3: Активовано значення налаштування положення'; 7587 'A07587 - Енкодер 1: Для попередньої обробки фактичного значення положення відсутній коректний енкодер'; 7588 'A07588 - Енкодер 2: Для попередньої обробки фактичного значення положення відсутній коректний енкодер'; 7589 'A07589 - Енкодер 3: Для попередньої обробки фактичного значення положення відсутній коректний енкодер'; 7590 'A07590 (F) - Енкодер 1: Виконується перемикання набору даних приводу'; 7591 'A07591 (F) - Енкодер 2: Виконується перемикання набору даних приводу'; 7592 'A07592 (F) - Енкодер 3: Виконується перемикання набору даних приводу'; 7593 'A07593 (F, N) - Енкодер 1: Перевищено діапазон значень фактичного положення'; 7594 'A07594 (F, N) - Енкодер 2: Перевищено діапазон значень фактичного положення'; 7595 'A07595 (F, N) - Енкодер 3: Перевищено діапазон значень фактичного положення'; 7596 'A07596 (F, N) - Енкодер 1: Функцію реферування перервано'; 7597 'A07597 (F, N) - Енкодер 2: Функцію реферування перервано'; 7598 'A07598 (F, N) - Енкодер 3: Функцію реферування перервано'; 7599 'F07599 (A) - Енкодер 1: Налаштування неможливе'; 7600 'F07600 (A) - Енкодер 2: Налаштування неможливе'; 7601 'F07601 (A) - Енкодер 3: Налаштування неможливе'; 7750 'F07750 - Привід: Параметр некоректний'; 7751 'F07751 - Привід: клапан не реагує'; 7752 'F07752 (A) - Привід: положення поршня неможливе'; 7753 'F07753 (N, A) - Привід: немає коректного фактичного значення тиску'; 7754 'F07754 - Привід: некоректна конфігурація запірного клапана'; 7755 'F07755 (N, A) - Привід: переміщення до жорсткого кінцевого упора без регулятора зусилля'; 7756 'F07756 - Привід: Фільтр власний частота > Найквіста частота'; 7800 'F07800 - Привід: силовий модуль відсутній'; 7801 'F07801 - Привід: Двигун Перевищення струму'; 7802 'F07802 - Привід: Ввід або Силовий модуль не готовий до роботи'; 7805 'A07805 (N) - Ввід: перевантаження I²t силового модуля'; 7807 'F07807 - Привід: виявлено коротке замикання/замикання на землю'; 7808 'F07808 (A) - Модуль ВЧ-демпфування: демпфування не готовий'; 7810 'F07810 - Привід: EEPROM силового модуля без номінальних даних'; 7815 'F07815 - Привід: силовий модуль замінено'; 7820 'A07820 - Привід: Температура датчик не підключено'; 7821 'A07821 - Контроль: швидкість опустилася нижче порога аварійного повідомлення'; 7822 'F07822 (N) - Контроль: швидкість опустилася нижче порога несправності'; 7823 'A07823 - I²t контроль аварійне повідомлення поріг перевищено'; 7824 'F07824 - I²t контроль несправність поріг перевищено'; 7825 'A07825 (N) - Привід: Симуляція режим активовано'; 7826 'F07826 - Привід: напруга кола постійного струму для режиму симуляції занадто висока'; 7840 'F07840 - Привід: Ввід робота відсутній'; 7841 'F07841 (A) - Привід: режим вводу скасовано'; 7850 'A07850 (F) - Зовнішній аварійне повідомлення 1'; 7851 'A07851 (F) - Зовнішній аварійне повідомлення 2'; 7852 'A07852 (F) - Зовнішній аварійне повідомлення 3'; 7860 'F07860 (A) - Зовнішній несправність 1'; 7861 'F07861 (A) - Зовнішній несправність 2'; 7862 'F07862 (A) - Зовнішній несправність 3'; 7890 'F07890 - Внутрішній захист напруги/внутрішнє коротке замикання якоря за активного STO'; 7898 'F07898 - Привід: підхоплення обертового двигуна не вдалося через надто малий потік'; 7899 'A07899 (N) - Привід: контроль заклинювання неможливий'; 7900 'F07900 (N, A) - Привід: заклинювання двигуна/регулятор швидкості на межі'; 7901 'F07901 - Привід: перевищення швидкості двигуна'; 7902 'F07902 (N, A) - Привід: двигун зупинився'; 7903 'A07903 - Привід: відхилення швидкості двигуна'; 7904 'F07904 (N, A) - Зовнішнє коротке замикання якоря: відсутній сигнал зворотного зв’язку контактора «Замкнено»'; 7905 'F07905 (N, A) - Зовнішній якір коротке замикання: Контактор зворотний зв’язок сигнал "Відкритий" відсутній'; 7906 'F07906 - Коротке замикання якоря/внутрішній захист напруги: помилка параметризації'; 7907 'F07907 - Внутрішнє коротке замикання якоря: після придушення імпульсів на клемах двигуна не нульовий потенціал'; 7908 'A07908 - Внутрішній якір коротке замикання активний'; 7909 'F07909 - Внутрішній захист напруги: деактивація діє лише після POWER ON'; 7910 'A07910 (N) - Привід: перегрів двигуна'; 7913 'F07913 - Збудження струм поза допуск діапазон'; 7914 'F07914 - Потік поза з допуск'; 7918 'A07918 (N) - Вибрано/активовано роботу трифазного генератора заданих значень'; 7920 'A07920 - Привід: крутний момент/швидкість занадто низькі'; 7921 'A07921 - Привід: крутний момент/швидкість занадто високі'; 7922 'A07922 - Привід: крутний момент/швидкість поза межами допуску'; 7923 'F07923 - Привід: крутний момент/швидкість занадто низькі'; 7924 'F07924 - Привід: крутний момент/швидкість занадто високі'; 7925 'F07925 - Привід: крутний момент/швидкість поза межами допуску'; 7926 'A07926 - Привід: некоректний параметр огинаючої кривої'; 7927 'A07927 - DC гальмівний активний'; 7928 'F07928 - Ініційовано внутрішній захист напруги'; 7930 'F07930 - Привід: Гальмо керування помилка'; 7931 'A07931 (F, N) - Гальмо виконує не відкритий'; 7932 'A07932 - Гальмо не загальмовується'; 7934 'F07934 (N) - Привід: конфігурація гальма утримання двигуна S120 Combi'; 7935 'F07935 (N) - Привід: Некоректний двигун утримання гальмо конфігурація'; 7937 'F07937 (N) - Привід: відхилення швидкості між моделлю двигуна та зовнішньою швидкістю'; 7940 'F07940 - Sync-line-drive: помилка синхронізації'; 7941 'A07941 - Sync-line-drive: задана частота не допускається'; 7942 'A07942 - Sync-line-drive: задана частота повністю відрізняється від цільової частоти'; 7943 'A07943 - Sync-line-drive: синхронізація не допускається'; 7950 'F07950 (A) - Привід: Некоректний двигун параметр'; 7955 'F07955 - Привід: Двигун має було змінено'; 7956 'F07956 (A) - Привід: код двигуна не відповідає двигуну зі списку (каталогу)'; 7960 'A07960 - Привід: Некоректний тертя характеристика'; 7961 'A07961 - Привід: активовано запис характеристики тертя'; 7963 'F07963 - Привід: запис характеристики тертя скасовано'; 7965 'A07965 (N) - Привід: Зберегти потрібно'; 7966 'F07966 - Привід: перевірте кут комутації'; 7967 'F07967 - Привід: некоректне автоматичне налаштування енкодера/ідентифікація положення полюса'; 7968 'F07968 - Привід: некоректне вимірювання Lq-Ld'; 7969 'F07969 - Привід: Некоректний полюс положення ідентифікація'; 7970 'F07970 - Привід: некоректне автоматичне налаштування енкодера'; 7971 'A07971 (N) - Привід: активовано визначення кутового зміщення комутації'; 7975 'A07975 (N) - Привід: Переміщення до нульовий мітка - задане вхід очікуваний'; 7976 'A07976 - Привід: активовано точне калібрування енкодера'; 7978 'A07978 (N) - Привід: активовано ESM режим очікує для кінець з двигун ідентифікація'; 7979 'A07979 (F, N) - Привід: полюс положення ідентифікація калібрування потрібно'; 7980 'A07980 - Привід: Обертовий вимірювання активовано'; 7981 'A07981 - Привід: Увімкнути сигнали для обертовий вимірювання відсутній'; 7982 'F07982 - Привід: Обертовий вимірювання енкодер тест'; 7983 'F07983 - Привід: характеристика насичення під час обертового вимірювання'; 7984 'F07984 - Привід: оптимізація регулятора швидкості, момент інерції'; 7985 'F07985 - Привід: оптимізація регулятора швидкості (коливальний тест)'; 7986 'F07986 - Привід: генератор рампової функції для обертового вимірювання'; 7987 'A07987 - Привід: Обертовий вимірювання, відсутній енкодер доступний'; 7988 'F07988 - Привід: Обертовий вимірювання, відсутній конфігурація вибрано'; 7989 'F07989 - Привід: індуктивність розсіювання під час обертового вимірювання (вісь q)'; 7990 'F07990 - Привід: Некоректний Ідентифікація даних двигуна'; 7991 'A07991 (N) - Привід: Ідентифікація даних двигуна активовано'; 7993 'F07993 - Привід: некоректний напрямок обертання поля або інверсія фактичного значення енкодера'; 7994 'A07994 (F, N) - Привід: ідентифікацію даних двигуна не виконано'; 7995 'F07995 - Привід: ідентифікація положення полюса не вдалася'; 7996 'F07996 - Привід: процедуру ідентифікації положення полюса не виконано'; 7998 'A07998 - Привід: ідентифікація даних двигуна активна на іншому приводі'; 7999 'A07999 - Привід: Ідентифікація даних двигуна не може бути активовано'; 8000 'F08000 (N, A) - TB: несправність живлення ±15 В'; 8010 'F08010 (N, A) - TB: аналого-цифровий перетворювач'; 8500 'F08500 (A) - COMM BOARD: Контроль час конфігурація закінчився'; 8501 'F08501 (N, A) - PN/COMM BOARD: тайм-аут заданого значення'; 8502 'F08502 (A) - PN/COMM BOARD: закінчився контрольний час сигналу справності'; 8504 'A08504 (F) - PN/COMM BOARD: Внутрішній Помилка циклічної передачі даних'; 8510 'F08510 (A) - PN/COMM BOARD: некоректні дані конфігурації передавання'; 8511 'A08511 (F) - PN/COMM BOARD: Приймання конфігурація дані некоректний'; 8520 'A08520 (F) - PN/COMM BOARD: помилка нециклічного каналу'; 8526 'A08526 (F) - PN/COMM BOARD: Відсутній циклічний з’єднання'; 8530 'A08530 (F) - PN/COMM BOARD: Повідомлення канал помилка'; 8531 'A08531 (F) - CBE20 POWER ON потрібно'; 8550 'A08550 - Помилка призначення апаратного інтерфейсу PZD'; 8555 'A08555 - Modbus TCP: помилка введення в експлуатацію'; 8560 'A08560 - IE: Синтаксис помилка у конфігурація файл'; 8561 'A08561 - IE: Узгодженість помилка що впливає на регульований параметри'; 8562 'A08562 - PROFINET: Синтаксис помилка у конфігурація файл'; 8563 'A08563 - PROFINET: Узгодженість помилка що впливає на регульований параметри'; 8564 'A08564 - PN/COMM BOARD: синтаксис помилка у конфігурація файл'; 8565 'A08565 - PNCOMM BOARD: Узгодженість помилка що впливає на регульований параметри'; 8700 'F08700 (A) - CAN: помилка зв’язку'; 8701 'F08701 - CAN: NMT стан зміна'; 8702 'F08702 (A) - CAN: RPDO Тайм-аут'; 8703 'F08703 (A) - CAN: Максимальний номер з привід об’єкти перевищено'; 8751 'A08751 (N) - CAN: втрата телеграми'; 8752 'A08752 - CAN: перевищено лічильник пасивних помилок'; 8753 'A08753 - CAN: переповнення буфера повідомлень'; 8754 'A08754 - CAN: некоректний режим зв’язку'; 8755 'A08755 - CAN: неможливо відобразити об’єкт'; 8756 'A08756 - CAN: перевищено кількість відображених байтів'; 8757 'A08757 - CAN: некоректний COB-ID'; 8758 'A08758 - CAN: Максимальний номер з коректний PDO перевищено'; 8759 'A08759 - CAN: PDO COB-ID вже доступний'; 8760 'A08760 - CAN: перевищено максимальний розмір IF PZD'; 8800 'A08800 - Активний енергозберігальний режим PROFIenergy'; 9000 'A09000 - Некоректно налаштовано користувача вебсервера'; 13000 'F13000 - Ліцензія не відповідає вимогам'; 13001 'A13001 - Помилка у ліцензія контрольна сума'; 13009 'F13009 - Ліцензування Технологія Розширення: ліцензія відсутня'; 13010 'F13010 - Ліцензійний функціональний модуль не ліцензовано'; 13020 'F13020 - Ліцензування не достатня у керування'; 13021 'A13021 - Відсутня ліцензія для вихідних частот > 550 Гц'; 13030 'A13030 - Пробний Ліцензія активовано'; 13031 'A13031 - Пробний Ліцензія період закінчився'; 13032 'A13032 - Активовано останній період пробної ліцензії'; 13033 'A13033 - Закінчився останній період пробної ліцензії'; 13100 'F13100 - Захист ноу-хау: помилка захисту від копіювання'; 13101 'F13101 - Захист ноу-хау: неможливо активувати захист від копіювання'; 13102 'F13102 - Захист ноу-хау: помилка узгодженості захищених даних'; 30001 'F30001 - Силовий модуль: перевищення струму'; 30002 'F30002 - Силовий модуль: перенапруга кола постійного струму'; 30003 'F30003 - Силовий модуль: занижена напруга кола постійного струму'; 30004 'F30004 - Силовий модуль: перегрів радіатора інвертора AC'; 30005 'F30005 - Силовий модуль: перевантаження I²t'; 30006 'F30006 - Силовий модуль: плата керування тиристорами'; 30008 'F30008 - Силовий модуль: помилка сигналу справності циклічних даних'; 30010 'A30010 (F) - Силовий модуль: помилка сигналу справності циклічних даних'; 30011 'F30011 - Силовий модуль: відсутня фаза мережі в головному колі'; 30012 'F30012 - Силовий модуль: обрив проводу датчика температури'; 30013 'F30013 - Силовий модуль: коротке замикання датчика температури'; 30015 'F30015 (N, A) - Силовий модуль: відсутня фаза кабелю двигуна'; 30016 'A30016 (N) - Силовий модуль: живлення навантаження вимкнено'; 30017 'F30017 - Силовий модуль: апаратне обмеження струму спрацьовувало надто часто'; 30020 'F30020 - Силовий модуль: конфігурація не підтримується'; 30021 'F30021 - Силовий модуль: замикання на землю'; 30022 'F30022 - Силовий модуль: контроль Uce'; 30024 'F30024 - Силовий модуль: перегрів за тепловою моделлю'; 30025 'F30025 - Силовий модуль: Перегрів кристала'; 30027 'F30027 - Силовий модуль: контроль часу попереднього заряду кола постійного струму'; 30030 'A30030 - Силовий модуль: внутрішній перегрів аварійне повідомлення'; 30031 'A30031 - Силовий модуль: апаратне обмеження струму у фазі U'; 30032 'A30032 - Силовий модуль: апаратне обмеження струму у фазі V'; 30033 'A30033 - Силовий модуль: апаратне обмеження струму у фазі W'; 30034 'A30034 - Силовий модуль: внутрішній перегрів'; 30035 'F30035 - Силовий модуль: перегрів повітря на вході'; 30036 'F30036 - Силовий модуль: внутрішній перегрів'; 30037 'F30037 - Силовий модуль: перегрів випрямляча'; 30038 'A30038 - Силовий модуль: контроль вентилятора конденсатора'; 30039 'F30039 - Силовий модуль: несправність вентилятора конденсатора'; 30040 'F30040 - Силовий модуль: занижена напруга 24 В'; 30041 'A30041 (F) - Силовий модуль: аварійне повідомлення про занижену напругу 24 В'; 30042 'A30042 - Силовий модуль: вентилятор досяг максимального напрацювання'; 30043 'F30043 - Силовий модуль: перенапруга 24 В'; 30044 'A30044 (F) - Силовий модуль: аварійне повідомлення про перенапругу 24 В'; 30045 'F30045 - Силовий модуль: Занижена напруга живлення'; 30046 'A30046 (F) - Силовий модуль: аварійне повідомлення про занижену напругу'; 30047 'F30047 - Охолоджувальний агрегат: Охолодження середовище витрата витрата занадто низький'; 30048 'A30048 (N) - Силовий модуль: несправний вентилятор'; 30049 'A30049 - Силовий модуль: несправний внутрішній вентилятор'; 30050 'F30050 - Силовий модуль: перенапруга живлення 24 В'; 30051 'F30051 - Силовий модуль: виявлено коротке замикання гальма утримання двигуна'; 30052 'F30052 - Помилка даних EEPROM'; 30053 'F30053 - FPGA дані несправний'; 30054 'A30054 (F, N) - Силовий модуль: занижена напруга під час розгальмовування гальма'; 30055 'F30055 - Силовий модуль: перевищення струму гальмівного переривника'; 30057 'A30057 - Силовий модуль: асиметрія мережі'; 30058 'F30058 (N, A) - Силовий модуль: несправний вентилятор радіатора'; 30059 'F30059 - Силовий модуль: несправний внутрішній вентилятор'; 30060 'F30060 (A) - Контроль стану контактора попереднього заряду'; 30061 'F30061 (A) - Контроль перемичкового контактора'; 30065 'A30065 (F, N) - Напруга виміряний значення не правдоподібний'; 30066 'A30066 (N) - Силовий модуль: аварійне повідомлення про перегрів конденсатора через повітряне охолодження'; 30067 'F30067 - Силовий модуль: несправність — перегрів конденсатора через повітряне охолодження'; 30068 'F30068 - Силовий модуль: знижена температура радіатора інвертора'; 30070 'F30070 - Цикл, запитаний силовим модулем, не підтримується'; 30071 'F30071 - Не отримано нових фактичних значень від силового модуля'; 30072 'F30072 - Задані значення більше не можуть передаватися до силового модуля'; 30073 'A30073 (N) - Попередня обробка фактичного/заданого значення більше не синхронна'; 30074 'F30074 (A) - Помилка зв’язку між Керування Модуль та Силовий модуль'; 30075 'F30075 - Не вдалося сконфігурувати силовий модуль'; 30076 'A30076 (N) - Силовий модуль: аварійне повідомлення про теплове перевантаження внутрішнього гальмівного резистора'; 30077 'A30077 (N) - Силовий модуль: теплове перевантаження внутрішнього гальмівного резистора'; 30078 'F30078 - Силовий модуль: несправний вентилятор або перегрів мережевого реактора'; 30079 'A30079 (N) - Силовий модуль: відносно напруги живлення напруга кола постійного струму занадто висока'; 30080 'F30080 - Силовий модуль: струм зростає надто швидко'; 30081 'F30081 - Силовий модуль: операції перемикання виконуються надто часто'; 30082 'A30082 - Силовий модуль: витрата охолоджувального середовища нижча за поріг аварійного повідомлення'; 30083 'F30083 - Силовий модуль: витрата охолоджувального середовища нижча за поріг несправності'; 30086 'A30086 - Силовий модуль: температура охолоджувальної рідини перевищила поріг аварійного повідомлення'; 30087 'F30087 - Силовий модуль: температура охолоджувальної рідини перевищила поріг несправності'; 30105 'F30105 - PU: несправність вимірювання фактичного значення'; 30314 'F30314 - Силовий модуль: живлення 24 В перевантажено PM'; 30315 'A30315 (F) - Силовий модуль: живлення 24 В перевантажено PM'; 30502 'A30502 - Силовий модуль: Перенапруга кола постійного струму'; 30600 'F30600 - SI P2: Ініційовано зупинку A'; 30611 'F30611 (A) - SI P2: Несправність у каналі контролю'; 30620 'N30620 (F, A) - SI P2: Безпечне вимкнення крутного моменту активний'; 30621 'N30621 (F, A) - SI P2: Активна безпечна зупинка 1'; 30625 'F30625 - SI P2: Помилка сигналу справності в даних безпеки'; 30630 'F30630 - SI P2: Гальмо керування помилка'; 30631 'F30631 - Керування гальмом: активне зовнішнє розгальмовування'; 30632 'F30632 - SI P2: Помилка сигналу керування/зворотного зв’язку запірного клапана'; 30640 'A30640 (F) - SI P2: несправність у тракті сигналу вимкнення другого каналу'; 30649 'F30649 - SI P2: Внутрішня програмна помилка'; 30650 'F30650 - SI P2: Потрібне приймальне випробування'; 30651 'F30651 - SI P2: не вдалося синхронізуватися з модулем керування'; 30652 'F30652 - SI P2: неприпустимий тактовий цикл контролю'; 30655 'F30655 - SI P2: Узгодьте функції контролю'; 30656 'F30656 - SI P2: Моторний модуль параметр помилка'; 30657 'F30657 - SI P2: Некоректний номер телеграми PROFIsafe'; 30659 'F30659 - SI P2: Запит на запис параметра відхилено'; 30664 'F30664 - Помилка під час завантаження'; 30665 'F30665 - SI P2: Система несправна'; 30666 'A30666 (F) - SI Motion P2: Постійний сигнал «1» на F-DI для безпечного квитування'; 30672 'F30672 - SI P2: Керування Модуль програмне забезпечення несумісний'; 30674 'F30674 - SI Motion P2: Функція безпеки не підтримується телеграмою PROFIsafe'; 30680 'F30680 - SI Motion P2: Помилка контрольної суми функцій контролю безпеки'; 30681 'F30681 - SI Motion P1: Некоректне значення параметра'; 30682 'F30682 - SI Motion P2: Функція контролю не підтримується'; 30683 'F30683 - SI Motion P2: Відсутній дозвіл SOS/SLS'; 30684 'F30684 - SI Motion P2: Граничні значення безпечно обмеженого положення переплутано'; 30685 'F30685 - SI Motion P2: Граничне значення безпечно обмеженої швидкості занадто високе'; 30686 'F30686 - SI Motion: Некоректна параметризація кулачкового положення'; 30688 'F30688 - SI Motion P2: Фактичний значення синхронізація не допустимий'; 30692 'F30692 - SI Motion P2: Значення параметра не допускається для режиму без енкодера'; 30693 'A30693 (F) - SI P2: змінено налаштування параметрів безпеки; потрібен теплий перезапуск/POWER ON'; 30700 'C30700 - SI Motion P2: Ініційовано зупинку A'; 30701 'C30701 - SI Motion P2: Ініційовано зупинку B'; 30706 'C30706 - SI Motion P2: Перевищено обмеження SAM/SBR'; 30707 'C30707 - SI Motion P2: Перевищено допуск для безпечної робочої зупинки'; 30708 'C30708 - SI Motion P2: Ініційовано зупинку C'; 30709 'C30709 - SI Motion P2: Ініційовано зупинку D'; 30710 'C30710 - SI Motion P2: Ініційовано зупинку E'; 30711 'C30711 - SI Motion P2: Несправність у каналі контролю'; 30712 'C30712 - SI Motion P2: Несправність обробки F-IO'; 30714 'C30714 - SI Motion P2: Безпечно обмежена швидкість перевищено'; 30715 'C30715 - SI Motion P2: Безпечно обмежене положення перевищено'; 30716 'C30716 - SI Motion P2: Перевищено допуск для безпечного напрямку руху'; 30717 'C30717 - SI Motion P2: Перевищено обмеження SLA'; 30730 'C30730 - SI Motion P2: Некоректний опорний блок для динамічної безпечно обмеженої швидкості'; 30770 'C30770 - SI Motion P2: Помилка розбіжності відмовобезпечних входів/виходів'; 30772 'A30772 - SI Motion P2: Виконується тестова зупинка для відмовобезпечних дискретних виходів'; 30773 'F30773 - SI Motion P2: Помилка тестової зупинки відмовобезпечного дискретного виходу'; 30788 'A30788 - Автоматичний тест зупинка: очікування для STO скасування вибору через SMM'; 30797 'C30797 - SI Motion P2: Вісь не пройшла безпечне реферування'; 30798 'C30798 - SI Motion P2: Тест зупинка для рух контроль функції виконується'; 30799 'C30799 - SI Motion P2: Приймальне тест режим активний'; 30800 'N30800 (F) - Силовий модуль: Груповий сигнал'; 30801 'F30801 - Силовий модуль DRIVE-CLiQ: відсутній сигнал справності'; 30802 'F30802 - Силовий модуль: Переповнення часового кванта'; 30804 'F30804 (N, A) - Силовий модуль: CRC'; 30805 'F30805 - Силовий модуль: Помилка контрольної суми EEPROM'; 30809 'F30809 - Силовий модуль: некоректна інформація про перемикання'; 30810 'A30810 (F) - Силовий модуль: сторожовий таймер'; 30820 'F30820 - Силовий модуль DRIVE-CLiQ: помилка телеграми'; 30835 'F30835 - Силовий модуль DRIVE-CLiQ: помилка циклічної передачі даних'; 30836 'F30836 - Силовий модуль DRIVE-CLiQ: помилка передавання даних DRIVE-CLiQ'; 30837 'F30837 - Силовий модуль DRIVE-CLiQ: несправність компонента'; 30845 'F30845 - Силовий модуль DRIVE-CLiQ: помилка циклічної передачі даних'; 30850 'F30850 - Силовий модуль: Внутрішня програмна помилка'; 30851 'F30851 - Силовий модуль DRIVE-CLiQ (CU): відсутній сигнал справності'; 30853 'A30853 - Силовий модуль: помилка сигналу справності циклічних даних'; 30860 'F30860 - Силовий модуль DRIVE-CLiQ (CU): помилка телеграми'; 30875 'F30875 - Силовий модуль: Несправність напруги живлення'; 30885 'F30885 - CU DRIVE-CLiQ (CU): помилка циклічної передачі даних'; 30886 'F30886 - PU DRIVE-CLiQ (CU): помилка під час передавання даних DRIVE-CLiQ'; 30887 'F30887 - Силовий модуль DRIVE-CLiQ (CU): несправність компонента'; 30895 'F30895 - PU DRIVE-CLiQ (CU): помилка почергової циклічної передачі даних'; 30896 'F30896 - Силовий модуль DRIVE-CLiQ (CU): некоректні властивості компонента'; 30899 'F30899 (N, A) - Силовий модуль: Невідома несправність'; 30903 'F30903 - Силовий модуль: Виникла помилка I2C-шини'; 30907 'F30907 - Силовий модуль: не вдалося сконфігурувати FPGA'; 30919 'A30919 - Силовий модуль: помилка контролю температури'; 30920 'A30920 (F) - Силовий модуль: несправність датчика температури'; 30930 'A30930 (N) - Силовий модуль: трасування компонента зберегло дані'; 30950 'F30950 - Силовий модуль: Внутрішня програмна помилка'; 30999 'A30999 (F, N) - Силовий модуль: Невідоме аварійне повідомлення'; 31100 'F31100 (N, A) - Енкодер 1: Помилка відстані до нульової мітки'; 31101 'F31101 (N, A) - Енкодер 1: Помилка нульової мітки'; 31103 'F31103 (N, A) - Енкодер 1: Сигнал рівень нульовий мітка (доріжка R) поза допуск'; 31110 'F31110 (N, A) - Енкодер 1: Помилка послідовного зв’язку'; 31111 'F31111 (N, A) - Енкодер 1: Енкодер сигналізує про внутрішню помилку (детальна інформація)'; 31112 'F31112 (N, A) - Енкодер 1: Енкодер сигналізує про внутрішню помилку'; 31115 'F31115 (N, A) - Енкодер 1: Рівень сигналу доріжки A або B занадто низький'; 31116 'F31116 (N, A) - Енкодер 1: Рівень сигналу доріжки A або B занадто низький'; 31117 'F31117 (N, A) - Енкодер 1: Помилка інверсії сигналів A/B/R'; 31118 'F31118 (N, A) - Енкодер 1: Зміна швидкості неправдоподібна'; 31120 'F31120 (N, A) - Енкодер 1: Несправність живлення енкодера'; 31121 'F31121 (N, A) - Енкодер 1: Некоректно визначено комутаційне положення'; 31122 'F31122 - Енкодер 1: Апаратна несправність модуля датчика'; 31123 'F31123 (N, A) - Енкодер 1: Рівень сигналу A/B поза межами допуску'; 31125 'F31125 (N, A) - Енкодер 1: Рівень сигналу доріжки A або B занадто високий'; 31126 'F31126 (N, A) - Енкодер 1: Рівень сигналу доріжки A або B занадто високий'; 31129 'F31129 (N, A) - Енкодер 1: Різниця положень датчика Холла/доріжок C/D та A/B занадто велика'; 31130 'F31130 (N, A) - Енкодер 1: Помилка нульової мітки та положення за грубою синхронізацією'; 31131 'F31131 (N, A) - Енкодер 1: Відхилення положення інкрементального/абсолютного енкодера занадто велике'; 31135 'F31135 - Енкодер 1: Помилка під час визначення положення (однообертовий режим)'; 31136 'F31136 - Енкодер 1: Помилка під час визначення положення (багатообертовий режим)'; 31137 'F31137 - Енкодер 1: Помилка під час визначення положення (однообертовий режим)'; 31138 'F31138 - Енкодер 1: Помилка під час визначення положення (багатообертовий режим)'; 31142 'F31142 (N, A) - Енкодер 1: Несправність напруги батареї'; 31150 'F31150 (N, A) - Енкодер 1: Помилка ініціалізації'; 31151 'F31151 (N, A) - Енкодер 1: Швидкість енкодера для ініціалізації AB занадто висока'; 31152 'F31152 (N, A) - Енкодер 1: Перевищено максимальну частоту сигналу (доріжка A/B)'; 31153 'F31153 (N, A) - Енкодер 1: Помилка ідентифікації'; 31160 'F31160 (N, A) - Енкодер 1: Несправність каналу A аналогового датчика'; 31161 'F31161 (N, A) - Енкодер 1: Несправність каналу B аналогового датчика'; 31163 'F31163 (N, A) - Енкодер 1: Значення положення аналогового датчика перевищує граничне значення'; 31400 'A31400 (F, N) - Енкодер 1: Помилка відстані до нульової мітки (перевищено поріг аварійного повідомлення)'; 31401 'A31401 (F, N) - Енкодер 1: Помилка нульової мітки (перевищено поріг аварійного повідомлення)'; 31405 'F31405 (N, A) - Енкодер 1: Перевищено температуру в модулі обробки сигналів енкодера'; 31407 'A31407 (F, N) - Енкодер 1: Досягнуто обмеження функції'; 31410 'A31410 (F, N) - Енкодер 1: Помилка зв’язку між енкодером і модулем датчика'; 31411 'A31411 (F, N) - Енкодер 1: Енкодер сигналізує про внутрішнє аварійне повідомлення (детальна інформація)'; 31412 'A31412 (F, N) - Енкодер 1: Енкодер сигналізує про внутрішнє аварійне повідомлення'; 31414 'A31414 (F, N) - Енкодер 1: Рівень сигналу доріжки C або D поза межами допуску'; 31415 'N31415 (F, A) - Енкодер 1: Рівень сигналу доріжки A або B поза межами допуску (аварійне повідомлення)'; 31418 'A31418 (F, N) - Енкодер 1: Зміна швидкості неправдоподібна (аварійне повідомлення)'; 31419 'A31419 (F, N) - Енкодер 1: Доріжка A або B поза межами допуску'; 31421 'A31421 (F, N) - Енкодер 1: Некоректно визначено комутаційне положення (аварійне повідомлення)'; 31422 'A31422 (F, N) - Енкодер 1: Імпульси на оберт прямокутний енкодер поза допуск смуга пропускання'; 31429 'A31429 (F, N) - Енкодер 1: Різниця положень датчика Холла/доріжок C/D та A/B занадто велика'; 31431 'A31431 (F, N) - Енкодер 1: Відхилення положення інкрементального/абсолютного енкодера занадто велике (аварійне повідомлення)'; 31432 'A31432 (F, N) - Енкодер 1: Адаптація положення ротора коригує відхилення'; 31442 'A31442 (F, N) - Енкодер 1: Досягнуто порога аварійного повідомлення за напругою батареї'; 31443 'A31443 (F, N) - Енкодер 1: Рівень сигналу доріжок C/D поза межами допуску (аварійне повідомлення)'; 31460 'A31460 (N) - Енкодер 1: Несправність каналу A аналогового датчика'; 31461 'A31461 (N) - Енкодер 1: Несправність каналу B аналогового датчика'; 31462 'A31462 (N) - Енкодер 1: Жоден канал аналогового датчика не активний'; 31463 'A31463 (N) - Енкодер 1: Значення положення аналогового датчика перевищує граничне значення'; 31470 'A31470 (F, N) - Енкодер 1: Енкодер сигналізує про внутрішню помилку (X521.7)'; 31500 'F31500 (N, A) - Енкодер 1: Перевищено діапазон переміщення для супроводження положення'; 31501 'F31501 (N, A) - Енкодер 1: Положення енкодера для супроводження положення поза межами вікна допуску'; 31502 'F31502 (N, A) - Енкодер 1: Енкодер із вимірювальною шестернею без коректних сигналів'; 31503 'F31503 (N, A) - Енкодер 1: Неможливо скинути супроводження положення'; 31700 'A31700 - Енкодер 1: ініційовано контроль функціональної безпеки'; 31800 'N31800 (F) - Енкодер 1: Груповий сигнал'; 31801 'F31801 (N, A) - Енкодер 1 DRIVE-CLiQ: відсутній сигнал справності'; 31802 'F31802 (N, A) - Енкодер 1: Переповнення часового кванта'; 31804 'F31804 (N, A) - Енкодер 1: Модуль датчика контрольна сума помилка'; 31805 'F31805 (N, A) - Енкодер 1: Помилка контрольної суми EEPROM'; 31806 'F31806 (N, A) - Енкодер 1: Помилка ініціалізації'; 31811 'A31811 (F, N) - Енкодер 1: Змінено серійний номер енкодера'; 31812 'F31812 (N, A) - Енкодер 1: Запитуваний цикл або синхронізація RX/TX не підтримується'; 31813 'F31813 - Енкодер 1: Несправність апаратного логічного модуля'; 31820 'F31820 (N, A) - Енкодер 1 DRIVE-CLiQ: помилка телеграми'; 31835 'F31835 (N, A) - Енкодер 1 DRIVE-CLiQ: помилка циклічної передачі даних'; 31836 'F31836 (N, A) - Енкодер 1 DRIVE-CLiQ: помилка передавання даних DRIVE-CLiQ'; 31837 'F31837 (N, A) - Енкодер 1 DRIVE-CLiQ: несправність компонента'; 31845 'F31845 (N, A) - Енкодер 1 DRIVE-CLiQ: помилка циклічної передачі даних'; 31850 'F31850 (N, A) - Енкодер 1: Внутрішня програмна помилка обробки сигналів енкодера'; 31851 'F31851 (N, A) - Енкодер 1 DRIVE-CLiQ (CU): відсутній сигнал справності'; 31860 'F31860 (N, A) - Енкодер 1 DRIVE-CLiQ (CU): помилка телеграми'; 31875 'F31875 (N, A) - Енкодер 1: Несправність напруги живлення'; 31885 'F31885 (N, A) - Енкодер 1 DRIVE-CLiQ (CU): помилка циклічної передачі даних'; 31886 'F31886 (N, A) - Енкодер 1 DRIVE-CLiQ (CU): помилка під час передавання даних DRIVE-CLiQ'; 31887 'F31887 (N, A) - Енкодер 1 DRIVE-CLiQ (CU): несправність компонента'; 31895 'F31895 (N, A) - Енкодер 1 DRIVE-CLiQ (CU): помилка почергової циклічної передачі даних'; 31896 'F31896 (N, A) - Енкодер 1 DRIVE-CLiQ (CU): некоректні властивості компонента'; 31899 'F31899 (N, A) - Енкодер 1: Невідома несправність'; 31902 'A31902 (F, N) - Енкодер 1: Виникла помилка SPI-шини'; 31903 'A31903 (F, N) - Енкодер 1: Виникла помилка I2C-шини'; 31905 'F31905 (N, A) - Енкодер 1: Помилка параметризації енкодера'; 31912 'F31912 - Енкодер 1: Комбінація пристроїв не допускається'; 31915 'A31915 (F, N) - Енкодер 1: Помилка конфігурації енкодера'; 31916 'F31916 (N, A) - Енкодер 1: Помилка параметризації енкодера'; 31920 'A31920 (F, N) - Енкодер 1: Температура датчик несправність (двигун)'; 31930 'A31930 (N) - Енкодер 1: Реєстратор даних зберіг дані'; 31940 'A31940 (F, N) - Енкодер 1: Некоректна напруга датчика шпинделя S1'; 31950 'F31950 - Енкодер 1: Внутрішня програмна помилка'; 31999 'A31999 (F, N) - Енкодер 1: Невідоме аварійне повідомлення'; 32100 'F32100 (N, A) - Енкодер 2: Помилка відстані до нульової мітки'; 32101 'F32101 (N, A) - Енкодер 2: Помилка нульової мітки'; 32103 'F32103 (N, A) - Енкодер 2: Сигнал рівень нульовий доріжка (доріжка R) поза допуск'; 32110 'F32110 (N, A) - Енкодер 2: Помилка послідовного зв’язку'; 32111 'F32111 (N, A) - Енкодер 2: Енкодер сигналізує про внутрішню помилку (детальна інформація)'; 32112 'F32112 (N, A) - Енкодер 2: Енкодер сигналізує про внутрішню помилку'; 32115 'F32115 (N, A) - Енкодер 2: Рівень сигналу доріжки A або B занадто низький'; 32116 'F32116 (N, A) - Енкодер 2: Рівень сигналу доріжки A або B занадто низький'; 32117 'F32117 (N, A) - Енкодер 2: Помилка інверсії сигналів A/B/R'; 32118 'F32118 (N, A) - Енкодер 2: Зміна швидкості неправдоподібна'; 32120 'F32120 (N, A) - Енкодер 2: Несправність живлення енкодера'; 32121 'F32121 (N, A) - Енкодер 2: Некоректно визначено комутаційне положення'; 32122 'F32122 - Енкодер 2: Апаратна несправність модуля датчика'; 32123 'F32123 (N, A) - Енкодер 2: Рівень сигналу A/B поза межами допуску'; 32125 'F32125 (N, A) - Енкодер 2: Рівень сигналу доріжки A або B занадто високий'; 32126 'F32126 (N, A) - Енкодер 2: Рівень сигналу доріжки A або B занадто високий'; 32129 'F32129 (N, A) - Енкодер 2: Різниця положень датчика Холла/доріжок C/D та A/B занадто велика'; 32130 'F32130 (N, A) - Енкодер 2: Помилка нульової мітки та положення за грубою синхронізацією'; 32131 'F32131 (N, A) - Енкодер 2: Відхилення положення інкрементального/абсолютного енкодера занадто велике'; 32135 'F32135 - Енкодер 2: Помилка під час визначення положення (однообертовий режим)'; 32136 'F32136 - Енкодер 2: Помилка під час визначення положення (багатообертовий режим)'; 32137 'F32137 - Енкодер 2: Помилка під час визначення положення (однообертовий режим)'; 32138 'F32138 - Енкодер 2: Помилка під час визначення положення (багатообертовий режим)'; 32142 'F32142 (N, A) - Енкодер 2: Несправність напруги батареї'; 32150 'F32150 (N, A) - Енкодер 2: Помилка ініціалізації'; 32151 'F32151 (N, A) - Енкодер 2: Швидкість енкодера для ініціалізації AB занадто висока'; 32152 'F32152 (N, A) - Енкодер 2: Перевищено максимальну частоту сигналу (доріжка A/B)'; 32153 'F32153 (N, A) - Енкодер 2: Помилка ідентифікації'; 32160 'F32160 (N, A) - Енкодер 2: Несправність каналу A аналогового датчика'; 32161 'F32161 (N, A) - Енкодер 2: Несправність каналу B аналогового датчика'; 32163 'F32163 (N, A) - Енкодер 2: Значення положення аналогового датчика перевищує граничне значення'; 32400 'A32400 (F, N) - Енкодер 2: Помилка відстані до нульової мітки (перевищено поріг аварійного повідомлення)'; 32401 'A32401 (F, N) - Енкодер 2: Помилка нульової мітки (перевищено поріг аварійного повідомлення)'; 32405 'F32405 (N, A) - Енкодер 2: Перевищено температуру в модулі обробки сигналів енкодера'; 32407 'A32407 (F, N) - Енкодер 2: Досягнуто обмеження функції'; 32410 'A32410 (F, N) - Енкодер 2: Помилка зв’язку між енкодером і модулем датчика'; 32411 'A32411 (F, N) - Енкодер 2: Енкодер сигналізує про внутрішнє аварійне повідомлення (детальна інформація)'; 32412 'A32412 (F, N) - Енкодер 2: Енкодер сигналізує про внутрішнє аварійне повідомлення'; 32414 'A32414 (F, N) - Енкодер 2: Рівень сигналу доріжки C або D поза межами допуску'; 32415 'N32415 (F, A) - Енкодер 2: Рівень сигналу доріжки A або B поза межами допуску (аварійне повідомлення)'; 32418 'A32418 (F, N) - Енкодер 2: Зміна швидкості неправдоподібна (аварійне повідомлення)'; 32419 'A32419 (F, N) - Енкодер 2: Доріжка A або B поза межами допуску'; 32421 'A32421 (F, N) - Енкодер 2: Некоректно визначено комутаційне положення (аварійне повідомлення)'; 32422 'A32422 (F, N) - Енкодер 2: Імпульси на оберт прямокутний енкодер поза допуск смуга пропускання'; 32429 'A32429 (F, N) - Енкодер 2: Різниця положень датчика Холла/доріжок C/D та A/B занадто велика'; 32431 'A32431 (F, N) - Енкодер 2: Відхилення положення інкрементального/абсолютного енкодера занадто велике (аварійне повідомлення)'; 32432 'A32432 (F, N) - Енкодер 2: Адаптація положення ротора коригує відхилення'; 32442 'A32442 (F, N) - Енкодер 2: Досягнуто порога аварійного повідомлення за напругою батареї'; 32443 'A32443 (F, N) - Енкодер 2: Рівень сигналу доріжок C/D поза межами допуску (аварійне повідомлення)'; 32460 'A32460 (N) - Енкодер 2: Несправність каналу A аналогового датчика'; 32461 'A32461 (N) - Енкодер 2: Несправність каналу B аналогового датчика'; 32462 'A32462 (N) - Енкодер 2: Жоден канал аналогового датчика не активний'; 32463 'A32463 (N) - Енкодер 2: Значення положення аналогового датчика перевищує граничне значення'; 32470 'A32470 (F, N) - Енкодер 2: Енкодер сигналізує про внутрішню помилку (X521.7)'; 32500 'F32500 (N, A) - Енкодер 2: Перевищено діапазон переміщення для супроводження положення'; 32501 'F32501 (N, A) - Енкодер 2: Положення енкодера для супроводження положення поза межами вікна допуску'; 32502 'F32502 (N, A) - Енкодер 2: Енкодер із вимірювальною шестернею без коректних сигналів'; 32503 'F32503 (N, A) - Енкодер 2: Неможливо скинути супроводження положення'; 32700 'A32700 - Енкодер 2: перевірка ефективності не дає очікуваного значення'; 32800 'N32800 (F) - Енкодер 2: Груповий сигнал'; 32801 'F32801 (N, A) - Енкодер 2 DRIVE-CLiQ: відсутній сигнал справності'; 32802 'F32802 (N, A) - Енкодер 2: Переповнення часового кванта'; 32804 'F32804 (N, A) - Енкодер 2: Модуль датчика контрольна сума помилка'; 32805 'F32805 (N, A) - Енкодер 2: Помилка контрольної суми EEPROM'; 32806 'F32806 (N, A) - Енкодер 2: Помилка ініціалізації'; 32811 'A32811 (F, N) - Енкодер 2: Змінено серійний номер енкодера'; 32812 'F32812 (N, A) - Енкодер 2: Запитуваний цикл або синхронізація RX/TX не підтримується'; 32813 'F32813 - Енкодер 2: Несправність апаратного логічного модуля'; 32820 'F32820 (N, A) - Енкодер 2 DRIVE-CLiQ: помилка телеграми'; 32835 'F32835 (N, A) - Енкодер 2 DRIVE-CLiQ: помилка циклічної передачі даних'; 32836 'F32836 (N, A) - Енкодер 2 DRIVE-CLiQ: помилка передавання даних DRIVE-CLiQ'; 32837 'F32837 (N, A) - Енкодер 2 DRIVE-CLiQ: несправність компонента'; 32845 'F32845 (N, A) - Енкодер 2 DRIVE-CLiQ: помилка циклічної передачі даних'; 32850 'F32850 (N, A) - Енкодер 2: Внутрішня програмна помилка обробки сигналів енкодера'; 32851 'F32851 (N, A) - Енкодер 2 DRIVE-CLiQ (CU): відсутній сигнал справності'; 32860 'F32860 (N, A) - Енкодер 2 DRIVE-CLiQ (CU): помилка телеграми'; 32875 'F32875 (N, A) - Енкодер 2: Несправність напруги живлення'; 32885 'F32885 (N, A) - Енкодер 2 DRIVE-CLiQ (CU): помилка циклічної передачі даних'; 32886 'F32886 (N, A) - Енкодер 2 DRIVE-CLiQ (CU): помилка під час передавання даних DRIVE-CLiQ'; 32887 'F32887 (N, A) - Енкодер 2 DRIVE-CLiQ (CU): несправність компонента'; 32895 'F32895 (N, A) - Енкодер 2 DRIVE-CLiQ (CU): помилка почергової циклічної передачі даних'; 32896 'F32896 (N, A) - Енкодер 2 DRIVE-CLiQ (CU): некоректні властивості компонента'; 32899 'F32899 (N, A) - Енкодер 2: Невідома несправність'; 32902 'A32902 (F, N) - Енкодер 2: Виникла помилка SPI-шини'; 32903 'A32903 (F, N) - Енкодер 2: Виникла помилка I2C-шини'; 32905 'F32905 (N, A) - Енкодер 2: Помилка параметризації енкодера'; 32912 'F32912 - Енкодер 2: Комбінація пристроїв не допускається'; 32915 'A32915 (F, N) - Енкодер 2: Помилка конфігурації енкодера'; 32916 'F32916 (N, A) - Енкодер 2: Помилка параметризації енкодера'; 32920 'A32920 (F, N) - Енкодер 2: Температура датчик несправність (двигун)'; 32930 'A32930 (N) - Енкодер 2: Реєстратор даних зберіг дані'; 32940 'A32940 (F, N) - Енкодер 2: Некоректна напруга датчика шпинделя S1'; 32950 'F32950 - Енкодер 2: Внутрішня програмна помилка'; 32999 'A32999 (F, N) - Енкодер 2: Невідоме аварійне повідомлення'; 33100 'F33100 (N, A) - Енкодер 3: Помилка відстані до нульової мітки'; 33101 'F33101 (N, A) - Енкодер 3: Помилка нульової мітки'; 33103 'F33103 (N, A) - Енкодер 3: Сигнал рівень нульовий доріжка (доріжка R) поза допуск'; 33110 'F33110 (N, A) - Енкодер 3: Помилка послідовного зв’язку'; 33111 'F33111 (N, A) - Енкодер 3: Енкодер сигналізує про внутрішню помилку (детальна інформація)'; 33112 'F33112 (N, A) - Енкодер 3: Енкодер сигналізує про внутрішню помилку'; 33115 'F33115 (N, A) - Енкодер 3: Рівень сигналу доріжки A або B занадто низький'; 33116 'F33116 (N, A) - Енкодер 3: Рівень сигналу доріжки A або B занадто низький'; 33117 'F33117 (N, A) - Енкодер 3: Помилка інверсії сигналів A/B/R'; 33118 'F33118 (N, A) - Енкодер 3: Зміна швидкості неправдоподібна'; 33120 'F33120 (N, A) - Енкодер 3: Несправність живлення енкодера'; 33121 'F33121 (N, A) - Енкодер 3: Некоректно визначено комутаційне положення'; 33122 'F33122 - Енкодер 3: Апаратна несправність модуля датчика'; 33123 'F33123 (N, A) - Енкодер 3: Рівень сигналу A/B поза межами допуску'; 33125 'F33125 (N, A) - Енкодер 3: Рівень сигналу доріжки A або B занадто високий'; 33126 'F33126 (N, A) - Енкодер 3: Рівень сигналу доріжки A або B занадто високий'; 33129 'F33129 (N, A) - Енкодер 3: Різниця положень датчика Холла/доріжок C/D та A/B занадто велика'; 33130 'F33130 (N, A) - Енкодер 3: Помилка нульової мітки та положення за грубою синхронізацією'; 33131 'F33131 (N, A) - Енкодер 3: Відхилення положення інкрементального/абсолютного енкодера занадто велике'; 33135 'F33135 - Енкодер 3: помилка під час визначення положення (однообертовий режим)'; 33136 'F33136 - Енкодер 3: Помилка під час визначення положення (багатообертовий режим)'; 33137 'F33137 - Енкодер 3: помилка під час визначення положення (однообертовий режим)'; 33138 'F33138 - Енкодер 3: Помилка під час визначення положення (багатообертовий режим)'; 33142 'F33142 (N, A) - Енкодер 3: Несправність напруги батареї'; 33150 'F33150 (N, A) - Енкодер 3: Помилка ініціалізації'; 33151 'F33151 (N, A) - Енкодер 3: Швидкість енкодера для ініціалізації AB занадто висока'; 33152 'F33152 (N, A) - Енкодер 3: Перевищено максимальну частоту сигналу (доріжка A/B)'; 33153 'F33153 (N, A) - Енкодер 3: Помилка ідентифікації'; 33160 'F33160 (N, A) - Енкодер 3: Несправність каналу A аналогового датчика'; 33161 'F33161 (N, A) - Енкодер 3: Несправність каналу B аналогового датчика'; 33163 'F33163 (N, A) - Енкодер 3: Значення положення аналогового датчика перевищує граничне значення'; 33400 'A33400 (F, N) - Енкодер 3: Помилка відстані до нульової мітки (перевищено поріг аварійного повідомлення)'; 33401 'A33401 (F, N) - Енкодер 3: Помилка нульової мітки (перевищено поріг аварійного повідомлення)'; 33405 'F33405 (N, A) - Енкодер 3: Перевищено температуру в модулі обробки сигналів енкодера'; 33407 'A33407 (F, N) - Енкодер 3: Досягнуто обмеження функції'; 33410 'A33410 (F, N) - Енкодер 3: Помилка зв’язку між енкодером і модулем датчика'; 33411 'A33411 (F, N) - Енкодер 3: Енкодер сигналізує про внутрішнє аварійне повідомлення (детальна інформація)'; 33412 'A33412 (F, N) - Енкодер 3: Енкодер сигналізує про внутрішнє аварійне повідомлення'; 33414 'A33414 (F, N) - Енкодер 3: Рівень сигналу доріжки C або D поза межами допуску'; 33415 'N33415 (F, A) - Енкодер 3: Рівень сигналу доріжки A або B поза межами допуску (аварійне повідомлення)'; 33418 'A33418 (F, N) - Енкодер 3: Зміна швидкості неправдоподібна (аварійне повідомлення)'; 33419 'A33419 (F, N) - Енкодер 3: Доріжка A або B поза межами допуску'; 33421 'A33421 (F, N) - Енкодер 3: Некоректно визначено комутаційне положення (аварійне повідомлення)'; 33422 'A33422 (F, N) - Енкодер 3: Імпульси на оберт прямокутний енкодер поза допуск смуга пропускання'; 33429 'A33429 (F, N) - Енкодер 3: Різниця положень датчика Холла/доріжок C/D та A/B занадто велика'; 33431 'A33431 (F, N) - Енкодер 3: Відхилення положення інкрементального/абсолютного енкодера занадто велике (аварійне повідомлення)'; 33432 'A33432 (F, N) - Енкодер 3: Адаптація положення ротора коригує відхилення'; 33442 'A33442 (F, N) - Енкодер 3: Досягнуто порога аварійного повідомлення за напругою батареї'; 33443 'A33443 (F, N) - Енкодер 3: Рівень сигналу доріжок C/D поза межами допуску (аварійне повідомлення)'; 33460 'A33460 (N) - Енкодер 3: Несправність каналу A аналогового датчика'; 33461 'A33461 (N) - Енкодер 3: Несправність каналу B аналогового датчика'; 33462 'A33462 (N) - Енкодер 3: Жоден канал аналогового датчика не активний'; 33463 'A33463 (N) - Енкодер 3: Значення положення аналогового датчика перевищує граничне значення'; 33470 'A33470 (F, N) - Енкодер 3: Енкодер сигналізує про внутрішню помилку (X521.7)'; 33500 'F33500 (N, A) - Енкодер 3: Перевищено діапазон переміщення для супроводження положення'; 33501 'F33501 (N, A) - Енкодер 3: Положення енкодера для супроводження положення поза межами вікна допуску'; 33502 'F33502 (N, A) - Енкодер 3: Енкодер із вимірювальною шестернею без коректних сигналів'; 33503 'F33503 (N, A) - Енкодер 3: Неможливо скинути супроводження положення'; 33700 'A33700 - Енкодер 3: перевірка ефективності не дає очікуваного значення'; 33800 'N33800 (F) - Енкодер 3: Груповий сигнал'; 33801 'F33801 (N, A) - Енкодер 3 DRIVE-CLiQ: відсутній сигнал справності'; 33802 'F33802 (N, A) - Енкодер 3: Переповнення часового кванта'; 33804 'F33804 (N, A) - Енкодер 3: Модуль датчика контрольна сума помилка'; 33805 'F33805 (N, A) - Енкодер 3: Помилка контрольної суми EEPROM'; 33806 'F33806 (N, A) - Енкодер 3: Помилка ініціалізації'; 33811 'A33811 (F, N) - Енкодер 3: Змінено серійний номер енкодера'; 33812 'F33812 (N, A) - Енкодер 3: Запитуваний цикл або синхронізація RX/TX не підтримується'; 33813 'F33813 - Енкодер 3: Несправність апаратного логічного модуля'; 33820 'F33820 (N, A) - Енкодер 3 DRIVE-CLiQ: помилка телеграми'; 33835 'F33835 (N, A) - Енкодер 3 DRIVE-CLiQ: помилка циклічної передачі даних'; 33836 'F33836 (N, A) - Енкодер 3 DRIVE-CLiQ: помилка передавання даних DRIVE-CLiQ'; 33837 'F33837 (N, A) - Енкодер 3 DRIVE-CLiQ: несправність компонента'; 33845 'F33845 (N, A) - Енкодер 3 DRIVE-CLiQ: помилка циклічної передачі даних'; 33850 'F33850 (N, A) - Енкодер 3: Внутрішня програмна помилка обробки сигналів енкодера'; 33851 'F33851 (N, A) - Енкодер 3 DRIVE-CLiQ (CU): відсутній сигнал справності'; 33860 'F33860 (N, A) - Енкодер 3 DRIVE-CLiQ (CU): помилка телеграми'; 33875 'F33875 (N, A) - Енкодер 3: Несправність напруги живлення'; 33885 'F33885 (N, A) - Енкодер 3 DRIVE-CLiQ (CU): помилка циклічної передачі даних'; 33886 'F33886 (N, A) - Енкодер 3 DRIVE-CLiQ (CU): помилка під час передавання даних DRIVE-CLiQ'; 33887 'F33887 (N, A) - Енкодер 3 DRIVE-CLiQ (CU): несправність компонента'; 33895 'F33895 (N, A) - Енкодер 3 DRIVE-CLiQ (CU): помилка почергової циклічної передачі даних'; 33896 'F33896 (N, A) - Енкодер 3 DRIVE-CLiQ (CU): некоректні властивості компонента'; 33899 'F33899 (N, A) - Енкодер 3: Невідома несправність'; 33902 'A33902 (F, N) - Енкодер 3: Виникла помилка SPI-шини'; 33903 'A33903 (F, N) - Енкодер 3: Виникла помилка I2C-шини'; 33905 'F33905 (N, A) - Енкодер 3: Помилка параметризації енкодера'; 33912 'F33912 - Енкодер 3: Комбінація пристроїв не допускається'; 33915 'A33915 (F, N) - Енкодер 3: Помилка конфігурації енкодера'; 33916 'F33916 (N, A) - Енкодер 3: Помилка параметризації енкодера'; 33920 'A33920 (F, N) - Енкодер 3: Температура датчик несправність (двигун)'; 33930 'A33930 (N) - Енкодер 3: Реєстратор даних зберіг дані'; 33940 'A33940 (F, N) - Енкодер 3: Некоректна напруга датчика шпинделя S1'; 33950 'F33950 - Енкодер 3: Внутрішня програмна помилка'; 33999 'A33999 (F, N) - Енкодер 3: Невідоме аварійне повідомлення'; 34207 'F34207 (N, A) - VSM: Перевищено поріг несправності за температурою'; 34211 'A34211 (F, N) - VSM: Перевищено поріг аварійного повідомлення за температурою'; 34800 'N34800 (F) - VSM: Груповий сигнал'; 34801 'F34801 (N, A) - VSM DRIVE-CLiQ: відсутній сигнал справності'; 34802 'F34802 (N, A) - VSM: Переповнення часового кванта'; 34803 'F34803 - VSM: Тест пам’яті'; 34804 'F34804 (N, A) - VSM: CRC'; 34805 'F34805 (N, A) - VSM: Помилка контрольної суми EEPROM'; 34806 'F34806 - VSM: Ініціалізація'; 34807 'A34807 (F, N) - VSM: Контроль часу керування послідовністю'; 34820 'F34820 - VSM DRIVE-CLiQ: помилка телеграми'; 34835 'F34835 - VSM DRIVE-CLiQ: помилка циклічної передачі даних'; 34836 'F34836 - VSM DRIVE-CLiQ: помилка передавання даних DRIVE-CLiQ'; 34837 'F34837 - VSM DRIVE-CLiQ: несправність компонента'; 34845 'F34845 - VSM DRIVE-CLiQ: помилка циклічної передачі даних'; 34850 'F34850 - VSM: Внутрішня програмна помилка'; 34851 'F34851 - VSM DRIVE-CLiQ (CU): відсутній сигнал справності'; 34860 'F34860 - VSM DRIVE-CLiQ (CU): помилка телеграми'; 34875 'F34875 - VSM: Несправність напруги живлення'; 34885 'F34885 - VSM DRIVE-CLiQ (CU): помилка циклічної передачі даних'; 34886 'F34886 - VSM DRIVE-CLiQ (CU): помилка під час передавання даних DRIVE-CLiQ'; 34887 'F34887 - VSM DRIVE-CLiQ (CU): несправність компонента'; 34895 'F34895 - VSM DRIVE-CLiQ (CU): помилка почергової циклічної передачі даних'; 34896 'F34896 - VSM DRIVE-CLiQ (CU): некоректні властивості компонента'; 34899 'F34899 (N, A) - VSM: Невідома несправність'; 34903 'A34903 (F, N) - VSM: Виникла помилка I2C-шини'; 34904 'A34904 (F, N) - VSM: EEPROM'; 34905 'A34905 (F, N) - VSM: Доступ до параметрів'; 34920 'F34920 (N, A) - VSM: Перегрів або несправність датчика температури'; 34950 'F34950 - VSM: Внутрішня програмна помилка'; 34999 'A34999 (F, N) - VSM: Невідоме аварійне повідомлення'; 35000 'F35000 - TM54F: Некоректний час дискретизації'; 35001 'F35001 - TM54F: Некоректне значення параметра'; 35002 'F35002 - TM54F: Введення в експлуатацію неможливе'; 35003 'F35003 - TM54F: Потрібне квитування на модулі керування'; 35004 'F35004 - TM54F: Некоректний цикл зв’язку'; 35005 'F35005 - TM54F:Паралельне з’єднання не підтримується'; 35006 'F35006 - TM54F: Некоректні групи приводів'; 35009 'F35009 - TM54F: Введення в експлуатацію функцій безпеки приводу не завершено'; 35011 'F35011 - TM54F: Призначення номера об’єкта приводу не допускається'; 35012 'A35012 - TM54F: Тестова зупинка для відмовобезпечних дискретних входів/виходів'; 35013 'F35013 - TM54F: Помилка тестової зупинки'; 35014 'A35014 - TM54F: Тестова зупинка для відмовобезпечних дискретних входів/виходів'; 35015 'A35015 - TM54F: моторний/гідравлічний модуль замінено або конфігурація некоректна'; 35016 'A35016 - TM54F: Мережевий обмін даними з приводом не встановлено'; 35040 'F35040 - TM54F: Занижена напруга 24 В'; 35043 'F35043 - TM54F: Перенапруга 24 В'; 35051 'F35051 - TM54F: Несправність у каналі контролю'; 35052 'F35052 (A) - TM54F: Внутрішня апаратна помилка'; 35053 'F35053 - TM54F: Перевищено поріг несправності за температурою'; 35054 'A35054 - TM54F: Перевищено поріг аварійного повідомлення за температурою'; 35075 'A35075 (F) - TM54F: Помилка внутрішнього зв’язку'; 35080 'A35080 (F) - TM54F: Помилка контрольної суми параметрів безпеки'; 35081 'A35081 (F) - TM54F: Постійний сигнал «1» на F-DI для безпечного квитування'; 35150 'F35150 - TM54F: Помилка зв’язку'; 35151 'F35151 - TM54F: Помилка розбіжності'; 35152 'F35152 - TM54F: Внутрішня програмна помилка'; 35200 'A35200 (F, N) - TM: дані калібрування'; 35207 'F35207 (N, A) - TM: Канал порога несправності/аварійного повідомлення за температурою 0 перевищено'; 35208 'F35208 (N, A) - TM: Канал порога несправності/аварійного повідомлення за температурою 1 перевищено'; 35209 'F35209 (N, A) - TM: Канал порога несправності/аварійного повідомлення за температурою 2 перевищено'; 35210 'F35210 (N, A) - TM: Канал порога несправності/аварійного повідомлення за температурою 3 перевищено'; 35211 'A35211 (F, N) - TM: Температура аварійне повідомлення поріг канал 0 перевищено'; 35212 'A35212 (F, N) - TM: Температура аварійне повідомлення поріг канал 1 перевищено'; 35213 'A35213 (F, N) - TM: Температура аварійне повідомлення поріг канал 2 перевищено'; 35214 'A35214 (F, N) - TM: Температура аварійне повідомлення поріг канал 3 перевищено'; 35220 'F35220 (N, A) - TM: Досягнуто обмеження частоти для сигнального виходу'; 35221 'F35221 (N, A) - TM: Відхилення між заданим і фактичним значеннями поза межами допуску'; 35222 'A35222 (F, N) - TM: Кількість імпульсів енкодера не допускається'; 35223 'A35223 (F, N) - TM: Зміщення нульової мітки не допускається'; 35224 'A35224 (N) - TM: Синхронізацію за нульовою міткою перервано'; 35225 'A35225 - TM: Синхронізацію за нульовою міткою утримано — енкодер не готовий до роботи'; 35226 'A35226 - TM: Доріжки A/B деактивовано'; 35227 'A35227 - Перемикання EDS/набору даних енкодера не підтримується'; 35228 'A35228 (F, N) - TM: некоректний час дискретизації p4099[3]'; 35229 'F35229 - TM: Часовий квант деактивовано'; 35230 'F35230 - TM: Апаратна несправність'; 35231 'A35231 - TM: Відсутнє головне керування від PLC'; 35232 'A35232 - TM41: Синхронізацію за нульовою міткою втрачено; потрібне повторне увімкнення живлення'; 35233 'F35233 - Функція компонента DRIVE-CLiQ не підтримується'; 35400 'F35400 (N, A) - TM: Канал порога несправності/аварійного повідомлення за температурою 4 перевищено'; 35401 'F35401 (N, A) - TM: Канал порога несправності/аварійного повідомлення за температурою 5 перевищено'; 35402 'F35402 (N, A) - TM: Канал порога несправності/аварійного повідомлення за температурою 6 перевищено'; 35403 'F35403 (N, A) - TM: Канал порога несправності/аварійного повідомлення за температурою 7 перевищено'; 35404 'F35404 (N, A) - TM: Канал порога несправності/аварійного повідомлення за температурою 8 перевищено'; 35405 'F35405 (N, A) - TM: Канал порога несправності/аварійного повідомлення за температурою 9 перевищено'; 35406 'F35406 (N, A) - TM: Канал порога несправності/аварійного повідомлення за температурою 10 перевищено'; 35407 'F35407 (N, A) - TM: Канал порога несправності/аварійного повідомлення за температурою 11 перевищено'; 35410 'A35410 (F, N) - TM: Температура аварійне повідомлення поріг канал 4 перевищено'; 35411 'A35411 (F, N) - TM: Температура аварійне повідомлення поріг канал 5 перевищено'; 35412 'A35412 (F, N) - TM: Температура аварійне повідомлення поріг канал 6 перевищено'; 35413 'A35413 (F, N) - TM: Температура аварійне повідомлення поріг канал 7 перевищено'; 35414 'A35414 (F, N) - TM: Температура аварійне повідомлення поріг канал 8 перевищено'; 35415 'A35415 (F, N) - TM: Температура аварійне повідомлення поріг канал 9 перевищено'; 35416 'A35416 (F, N) - TM: Температура аварійне повідомлення поріг канал 10 перевищено'; 35417 'A35417 (F, N) - TM: Температура аварійне повідомлення поріг канал 11 перевищено'; 35800 'N35800 (F) - TM: Груповий сигнал'; 35801 'F35801 (N, A) - TM DRIVE-CLiQ: відсутній сигнал справності'; 35802 'A35802 (F, N) - TM: Переповнення часового кванта'; 35803 'A35803 (F, N) - TM: Тест пам’яті'; 35804 'F35804 (N, A) - TM: CRC'; 35805 'F35805 (N, A) - TM: Помилка контрольної суми EEPROM'; 35807 'A35807 (F, N) - TM: Контроль часу керування послідовністю'; 35820 'F35820 - TM DRIVE-CLiQ: помилка телеграми'; 35835 'F35835 - TM DRIVE-CLiQ: помилка циклічної передачі даних'; 35836 'F35836 - TM DRIVE-CLiQ: помилка передавання даних DRIVE-CLiQ'; 35837 'F35837 - PTM DRIVE-CLiQ: несправність компонента'; 35845 'F35845 - TM DRIVE-CLiQ: помилка циклічної передачі даних'; 35850 'F35850 - TM: Внутрішня програмна помилка'; 35851 'F35851 - TM DRIVE-CLiQ (CU): відсутній сигнал справності'; 35860 'F35860 - TM DRIVE-CLiQ (CU): помилка телеграми'; 35875 'F35875 - TM: Несправність напруги живлення'; 35885 'F35885 - TM DRIVE-CLiQ (CU): помилка циклічної передачі даних'; 35886 'F35886 - TM DRIVE-CLiQ (CU): помилка під час передавання даних DRIVE-CLiQ'; 35887 'F35887 - TM DRIVE-CLiQ (CU): несправність компонента'; 35895 'F35895 - TM DRIVE-CLiQ (CU): помилка почергової циклічної передачі даних'; 35896 'F35896 - TM DRIVE-CLiQ (CU): некоректні властивості компонента'; 35899 'F35899 (N, A) - TM: Невідома несправність'; 35903 'A35903 (F, N) - TM: Виникла помилка I2C-шини'; 35904 'A35904 (F, N) - TM: EEPROM'; 35905 'A35905 (F, N) - TM: Доступ до параметрів'; 35906 'A35906 (F, N) - TM: Відсутнє живлення 24 В'; 35907 'A35907 (F, N) - TM: Помилка ініціалізації обладнання'; 35910 'A35910 (F, N) - TM: Перегрів модуля'; 35911 'A35911 (F, N) - TM: Годинник синхронний робота Відсутній сигнал справності'; 35920 'A35920 (F, N) - TM: Помилка каналу датчика температури 0'; 35921 'A35921 (F, N) - TM: Помилка каналу датчика температури 1'; 35922 'A35922 (F, N) - TM: Помилка каналу датчика температури 2'; 35923 'A35923 (F, N) - TM: Помилка каналу датчика температури 3'; 35924 'A35924 (F, N) - TM: Помилка каналу датчика температури 4'; 35925 'A35925 (F, N) - TM: Помилка каналу датчика температури 5'; 35926 'A35926 (F, N) - TM: Помилка каналу датчика температури 6'; 35927 'A35927 (F, N) - TM: Помилка каналу датчика температури 7'; 35928 'A35928 (F, N) - TM: Помилка каналу датчика температури 8'; 35929 'A35929 (F, N) - TM: Помилка каналу датчика температури 9'; 35930 'A35930 (F, N) - TM: Помилка каналу датчика температури 10'; 35931 'A35931 (F, N) - TM: Помилка каналу датчика температури 11'; 35950 'F35950 - TM: Внутрішня програмна помилка'; 35999 'A35999 (F, N) - TM: Невідоме аварійне повідомлення'; 36207 'F36207 (N, A) - Hub: Перегрів компонента'; 36211 'A36211 (F, N) - Hub: Аварійне повідомлення про перегрів компонента'; 36214 'F36214 (N, A) - Hub: несправність — перенапруга живлення 24 В'; 36216 'F36216 (N, A) - Hub: несправність — занижена напруга живлення 24 В'; 36217 'A36217 (N) - Hub: аварійне повідомлення про занижену напругу живлення 24 В'; 36800 'N36800 (F) - Hub: Груповий сигнал'; 36801 'A36801 (F, N) - Hub DRIVE-CLiQ: відсутній сигнал справності'; 36802 'A36802 (F, N) - Hub: Переповнення часового кванта'; 36804 'F36804 (N, A) - Hub: Контрольна сума помилка'; 36805 'F36805 (N, A) - Hub: Некоректна контрольна сума EEPROM'; 36820 'F36820 - Hub DRIVE-CLiQ: помилка телеграми'; 36835 'F36835 - Hub DRIVE-CLiQ: помилка циклічної передачі даних'; 36836 'F36836 - Hub DRIVE-CLiQ: помилка передавання даних DRIVE-CLiQ'; 36837 'F36837 - Hub DRIVE-CLiQ: несправність компонента'; 36845 'F36845 - Hub DRIVE-CLiQ: помилка циклічної передачі даних'; 36851 'F36851 - Hub DRIVE-CLiQ (CU): відсутній сигнал справності'; 36860 'F36860 - Hub DRIVE-CLiQ (CU): помилка телеграми'; 36875 'F36875 - HUB: Несправність напруги живлення'; 36885 'F36885 - Hub DRIVE-CLiQ (CU): помилка циклічної передачі даних'; 36886 'F36886 - Hub DRIVE-CLiQ (CU): помилка під час передавання даних DRIVE-CLiQ'; 36887 'F36887 - Hub DRIVE-CLiQ (CU): несправність компонента'; 36895 'F36895 - Hub DRIVE-CLiQ (CU): помилка почергової циклічної передачі даних'; 36896 'F36896 - Hub DRIVE-CLiQ (CU): некоректні властивості компонента'; 36899 'F36899 (N, A) - Hub: Невідома несправність'; 36950 'F36950 - Hub: Внутрішня програмна помилка'; 36999 'A36999 (F, N) - Hub: Невідоме аварійне повідомлення'; 37001 'F37001 - Модуль ВЧ-демпфування: Перевищення струму'; 37002 'F37002 - Модуль ВЧ-демпфування: Напруга демпфування занадто висока'; 37003 'F37003 - Модуль ВЧ-демпфування: Напругу демпфування не встановлено'; 37004 'F37004 - Модуль ВЧ-демпфування: Перегрів радіатора'; 37005 'F37005 - Модуль ВЧ-демпфування: Перевантаження I²t'; 37012 'F37012 - Модуль ВЧ-демпфування: Обрив проводу датчика температури радіатора'; 37013 'F37013 - Модуль ВЧ-демпфування: Коротке замикання датчика температури радіатора'; 37024 'F37024 - Модуль ВЧ-демпфування: Перегрів за тепловою моделлю'; 37025 'F37025 - Модуль ВЧ-демпфування: Перегрів кристала'; 37034 'A37034 - Модуль ВЧ-демпфування: Внутрішній перегрів'; 37036 'F37036 - Модуль ВЧ-демпфування: Внутрішній перегрів'; 37040 'F37040 - Модуль ВЧ-демпфування: Занижена напруга 24 В'; 37041 'A37041 (F) - Модуль ВЧ-демпфування: Аварійне повідомлення про занижену напругу 24 В'; 37043 'F37043 - Модуль ВЧ-демпфування: Перенапруга 24 В'; 37044 'A37044 (F) - Модуль ВЧ-демпфування: Аварійне повідомлення про перенапругу 24 В'; 37045 'F37045 - Модуль ВЧ-демпфування: Занижена напруга живлення'; 37049 'A37049 - Модуль ВЧ-демпфування: Несправний внутрішній вентилятор'; 37050 'F37050 